LIN {X 0,Y 383.942,Z 862.362,A -85,B 0,C 180,E1 18991.194,E2 18991.194} C_VEL
LIN {X 0,Y 383.942,Z 862.362,A -85,B 0,C 180,E1 18988.806,E2 18988.806} C_VEL
LIN {X 0,Y 383.936,Z 861.248,A -85,B 0,C 180,E1 18986.267,E2 18986.267} C_VEL
LIN {X 0,Y 383.976,Z 858.254,A -85,B 0,C 180,E1 18983.121,E2 18983.121} C_VEL
LIN {X 0,Y 384.141,Z 854.129,A -85,B 0,C 180,E1 18980.411,E2 18980.411} C_VEL
LIN {X 0,Y 384.492,Z 848.967,A -85,B 0,C 180,E1 18977.841,E2 18977.841} C_VEL
LIN {X 0,Y 385.264,Z 841.518,A -85,B 0,C 180,E1 18974.901,E2 18974.901} C_VEL
LIN {X 0,Y 386.443,Z 832.341,A -85,B 0,C 180,E1 18972.068,E2 18972.068} C_VEL
LIN {X 0,Y 387.786,Z 823.59,A -85,B 0,C 180,E1 18969.788,E2 18969.788} C_VEL
LIN {X 0,Y 389.798,Z 811.997,A -85,B 0,C 180,E1 18967.213,E2 18967.213} C_VEL
LIN {X 0,Y 392.168,Z 798.843,A -85,B 0,C 180,E1 18964.801,E2 18964.801} C_VEL
LIN {X 0,Y 394.491,Z 786.516,A -85,B 0,C 180,E1 18962.857,E2 18962.857} C_VEL
LIN {X 0,Y 397.519,Z 770.561,A -85,B 0,C 180,E1 18960.712,E2 18960.712} C_VEL
LIN {X 0,Y 400.36,Z 754.684,A -85,B 0,C 180,E1 18958.943,E2 18958.943} C_VEL
LIN {X 0,Y 402.909,Z 739.928,A -85,B 0,C 180,E1 18957.543,E2 18957.543} C_VEL
LIN {X 0,Y 405.855,Z 721.57,A -85,B 0,C 180,E1 18956.083,E2 18956.083} C_VEL
LIN {X 0,Y 408.29,Z 703.761,A -85,B 0,C 180,E1 18954.953,E2 18954.953} C_VEL
LIN {X 0,Y 410.239,Z 687.519,A -85,B 0,C 180,E1 18954.116,E2 18954.116} C_VEL
LIN {X 0,Y 412.235,Z 667.836,A -85,B 0,C 180,E1 18953.326,E2 18953.326} C_VEL
LIN {X 0,Y 413.644,Z 647.128,A -85,B 0,C 180,E1 18952.766,E2 18952.766} C_VEL
LIN {X 0,Y 420.093,Z 444.232,A -85,B 0,C 180,E1 18949.037,E2 18949.037} C_VEL
LIN {X 0,Y 418.812,Z 440.206,A -85,B 0,C 180,E1 18948.796,E2 18948.796} C_VEL
LIN {X 0,Y 408.36,Z 420.188,A -85,B 0,C 180,E1 18947.041,E2 18947.041} C_VEL
LIN {X 0,Y 398.971,Z 403.892,A -85,B 0,C 180,E1 18945.381,E2 18945.381} C_VEL
LIN {X 0,Y 391.846,Z 392.481,A -85,B 0,C 180,E1 18944.058,E2 18944.058} C_VEL
LIN {X 0,Y 389.279,Z 388.042,A -85,B 0,C 180,E1 18943.505,E2 18943.505} C_VEL
LIN {X 0,Y 385.572,Z 377.041,A -85,B 0,C 180,E1 18940.395,E2 18940.395} C_VEL
LIN {X 0,Y 385.574,Z 376.942,A -85,B 0,C 180,E1 18936.619,E2 18936.619} C_VEL
LIN {X 0,Y 385.58,Z 376.931,A -85,B 0,C 180,E1 18932.646,E2 18932.646} C_VEL
LIN {X 0,Y 385.598,Z 376.915,A -85,B 0,C 180,E1 18928.788,E2 18928.788} C_VEL
LIN {X 0,Y 385.593,Z 376.956,A -85,B 0,C 180,E1 18924.681,E2 18924.681} C_VEL
LIN {X 0,Y 385.592,Z 376.909,A -85,B 0,C 180,E1 18920.655,E2 18920.655} C_VEL
LIN {X 0,Y 385.593,Z 376.941,A -85,B 0,C 180,E1 18916.578,E2 18916.578} C_VEL
LIN {X 0,Y 385.593,Z 376.919,A -85,B 0,C 180,E1 18912.586,E2 18912.586} C_VEL
LIN {X 0,Y 385.597,Z 376.93,A -85,B 0,C 180,E1 18908.505,E2 18908.505} C_VEL
LIN {X 0,Y 385.591,Z 376.927,A -85,B 0,C 180,E1 18904.468,E2 18904.468} C_VEL
LIN {X 0,Y 385.605,Z 376.925,A -85,B 0,C 180,E1 18900.452,E2 18900.452} C_VEL
LIN {X 0,Y 385.591,Z 376.927,A -85,B 0,C 180,E1 18896.439,E2 18896.439} C_VEL
LIN {X 0,Y 385.601,Z 376.923,A -85,B 0,C 180,E1 18892.408,E2 18892.408} C_VEL
LIN {X 0,Y 385.592,Z 376.934,A -85,B 0,C 180,E1 18888.338,E2 18888.338} C_VEL
LIN {X 0,Y 385.589,Z 376.916,A -85,B 0,C 180,E1 18884.363,E2 18884.363} C_VEL
LIN {X 0,Y 385.595,Z 376.946,A -85,B 0,C 180,E1 18880.261,E2 18880.261} C_VEL
LIN {X 0,Y 385.581,Z 376.911,A -85,B 0,C 180,E1 18876.31,E2 18876.31} C_VEL
LIN {X 0,Y 385.578,Z 376.958,A -85,B 0,C 180,E1 18872.353,E2 18872.353} C_VEL
LIN {X 0,Y 385.562,Z 376.958,A -85,B 0,C 180,E1 18868.556,E2 18868.556} C_VEL
LIN {X 0,Y 385.554,Z 376.96,A -85,B 0,C 180,E1 18864.679,E2 18864.679} C_VEL
LIN {X 0,Y 385.55,Z 376.957,A -85,B 0,C 180,E1 18860.757,E2 18860.757} C_VEL
LIN {X 0,Y 385.553,Z 376.96,A -85,B 0,C 180,E1 18856.777,E2 18856.777} C_VEL
LIN {X 0,Y 385.553,Z 376.96,A -85,B 0,C 180,E1 18852.799,E2 18852.799} C_VEL
LIN {X 0,Y 385.554,Z 376.956,A -85,B 0,C 180,E1 18848.87,E2 18848.87} C_VEL
LIN {X 0,Y 385.56,Z 376.957,A -85,B 0,C 180,E1 18844.966,E2 18844.966} C_VEL
LIN {X 0,Y 385.568,Z 376.959,A -85,B 0,C 180,E1 18841.067,E2 18841.067} C_VEL
LIN {X 0,Y 385.579,Z 376.954,A -85,B 0,C 180,E1 18837.154,E2 18837.154} C_VEL
LIN {X 0,Y 385.628,Z 377.162,A -85,B 0,C 180,E1 18833.371,E2 18833.371} C_VEL
LIN {X 0,Y 386.073,Z 378.926,A -85,B 0,C 180,E1 18831.816,E2 18831.816} C_VEL
LIN {X 0,Y 387.404,Z 381.16,A -85,B 0,C 180,E1 18830.07,E2 18830.07} C_VEL
LIN {X 0,Y 389.591,Z 382.927,A -85,B 0,C 180,E1 18827.165,E2 18827.165} C_VEL
LIN {X 0,Y 391.833,Z 384.088,A -85,B 0,C 180,E1 18823.728,E2 18823.728} C_VEL
LIN {X 0,Y 393.13,Z 386.138,A -85,B 0,C 180,E1 18820.996,E2 18820.996} C_VEL
LIN {X 0,Y 394.172,Z 387.9,A -85,B 0,C 180,E1 18818.166,E2 18818.166} C_VEL
LIN {X 0,Y 395.064,Z 388.811,A -85,B 0,C 180,E1 18814.791,E2 18814.791} C_VEL
LIN {X 0,Y 395.484,Z 389.178,A -85,B 0,C 180,E1 18811.449,E2 18811.449} C_VEL
LIN {X 0,Y 395.444,Z 389.163,A -85,B 0,C 180,E1 18808.116,E2 18808.116} C_VEL
LIN {X 0,Y 394.988,Z 388.728,A -85,B 0,C 180,E1 18804.917,E2 18804.917} C_VEL
LIN {X 0,Y 394.109,Z 387.826,A -85,B 0,C 180,E1 18801.686,E2 18801.686} C_VEL
LIN {X 0,Y 393.123,Z 386.118,A -85,B 0,C 180,E1 18798.98,E2 18798.98} C_VEL
LIN {X 0,Y 391.832,Z 384.088,A -85,B 0,C 180,E1 18796.272,E2 18796.272} C_VEL
LIN {X 0,Y 389.591,Z 382.928,A -85,B 0,C 180,E1 18792.835,E2 18792.835} C_VEL
LIN {X 0,Y 387.4,Z 381.156,A -85,B 0,C 180,E1 18789.925,E2 18789.925} C_VEL
LIN {X 0,Y 386.016,Z 378.794,A -85,B 0,C 180,E1 18788.101,E2 18788.101} C_VEL
LIN {X 0,Y 385.613,Z 377.094,A -85,B 0,C 180,E1 18786.51,E2 18786.51} C_VEL
LIN {X 0,Y 385.593,Z 376.953,A -85,B 0,C 180,E1 18782.651,E2 18782.651} C_VEL
LIN {X 0,Y 384.623,Z 377.077,A -85,B 0,C 180,E1 18781.507,E2 18781.507} C_VEL
LIN {X 0,Y 379.656,Z 377.695,A -85,B 0,C 180,E1 18779.185,E2 18779.185} C_VEL
LIN {X 0,Y 377.705,Z 377.936,A -85,B 0,C 180,E1 18777.774,E2 18777.774} C_VEL
LIN {X 0,Y 377.612,Z 377.948,A -85,B 0,C 180,E1 18777.434,E2 18777.434} C_VEL
LIN {X 0,Y 377.613,Z 377.947,A -85,B 0,C 180,E1 18773.333,E2 18773.333} C_VEL
LIN {X 0,Y 377.611,Z 377.946,A -85,B 0,C 180,E1 18769.356,E2 18769.356} C_VEL
LIN {X 0,Y 377.613,Z 377.95,A -85,B 0,C 180,E1 18765.227,E2 18765.227} C_VEL
LIN {X 0,Y 377.612,Z 377.947,A -85,B 0,C 180,E1 18761.235,E2 18761.235} C_VEL
LIN {X 0,Y 377.615,Z 377.945,A -85,B 0,C 180,E1 18757.124,E2 18757.124} C_VEL
LIN {X 0,Y 377.614,Z 377.949,A -85,B 0,C 180,E1 18753.045,E2 18753.045} C_VEL
LIN {X 0,Y 377.616,Z 377.947,A -85,B 0,C 180,E1 18748.973,E2 18748.973} C_VEL
LIN {X 0,Y 377.61,Z 377.907,A -85,B 0,C 180,E1 18744.889,E2 18744.889} C_VEL
LIN {X 0,Y 377.615,Z 377.947,A -85,B 0,C 180,E1 18740.773,E2 18740.773} C_VEL
LIN {X 0,Y 377.608,Z 377.895,A -85,B 0,C 180,E1 18736.767,E2 18736.767} C_VEL
LIN {X 0,Y 377.613,Z 377.947,A -85,B 0,C 180,E1 18732.688,E2 18732.688} C_VEL
LIN {X 0,Y 377.609,Z 377.896,A -85,B 0,C 180,E1 18728.673,E2 18728.673} C_VEL
LIN {X 0,Y 377.615,Z 377.94,A -85,B 0,C 180,E1 18724.549,E2 18724.549} C_VEL
LIN {X 0,Y 377.609,Z 377.899,A -85,B 0,C 180,E1 18720.449,E2 18720.449} C_VEL
LIN {X 0,Y 377.614,Z 377.941,A -85,B 0,C 180,E1 18716.502,E2 18716.502} C_VEL
LIN {X 0,Y 377.609,Z 377.901,A -85,B 0,C 180,E1 18712.386,E2 18712.386} C_VEL
LIN {X 0,Y 377.616,Z 377.933,A -85,B 0,C 180,E1 18708.385,E2 18708.385} C_VEL
LIN {X 0,Y 377.614,Z 377.91,A -85,B 0,C 180,E1 18704.325,E2 18704.325} C_VEL
LIN {X 0,Y 377.615,Z 377.918,A -85,B 0,C 180,E1 18700.344,E2 18700.344} C_VEL
LIN {X 0,Y 377.617,Z 377.936,A -85,B 0,C 180,E1 18696.262,E2 18696.262} C_VEL
LIN {X 0,Y 377.613,Z 377.902,A -85,B 0,C 180,E1 18692.172,E2 18692.172} C_VEL
LIN {X 0,Y 377.621,Z 377.935,A -85,B 0,C 180,E1 18688.198,E2 18688.198} C_VEL
LIN {X 0,Y 377.62,Z 377.947,A -85,B 0,C 180,E1 18684.115,E2 18684.115} C_VEL
LIN {X 0,Y 377.681,Z 378.167,A -85,B 0,C 180,E1 18680.625,E2 18680.625} C_VEL
LIN {X 0,Y 381.123,Z 388.069,A -85,B 0,C 180,E1 18677.756,E2 18677.756} C_VEL
LIN {X 0,Y 390.405,Z 402.884,A -85,B 0,C 180,E1 18675.89,E2 18675.89} C_VEL
LIN {X 0,Y 399.613,Z 418.325,A -85,B 0,C 180,E1 18674.175,E2 18674.175} C_VEL
LIN {X 0,Y 409.795,Z 437.296,A -85,B 0,C 180,E1 18672.376,E2 18672.376} C_VEL
LIN {X 0,Y 414.001,Z 446.197,A -85,B 0,C 180,E1 18671.649,E2 18671.649} C_VEL
LIN {X 0,Y 407.264,Z 647.302,A -85,B 0,C 180,E1 18667.908,E2 18667.908} C_VEL
LIN {X 0,Y 405.749,Z 668.252,A -85,B 0,C 180,E1 18667.327,E2 18667.327} C_VEL
LIN {X 0,Y 403.735,Z 687.281,A -85,B 0,C 180,E1 18666.554,E2 18666.554} C_VEL
LIN {X 0,Y 401.698,Z 703.522,A -85,B 0,C 180,E1 18665.709,E2 18665.709} C_VEL
LIN {X 0,Y 399,Z 722.359,A -85,B 0,C 180,E1 18664.494,E2 18664.494} C_VEL
LIN {X 0,Y 395.936,Z 740.419,A -85,B 0,C 180,E1 18663.023,E2 18663.023} C_VEL
LIN {X 0,Y 393.241,Z 755.268,A -85,B 0,C 180,E1 18661.585,E2 18661.585} C_VEL
LIN {X 0,Y 390.053,Z 772.125,A -85,B 0,C 180,E1 18659.651,E2 18659.651} C_VEL
LIN {X 0,Y 387.116,Z 786.716,A -85,B 0,C 180,E1 18657.63,E2 18657.63} C_VEL
LIN {X 0,Y 384.752,Z 798.6,A -85,B 0,C 180,E1 18655.72,E2 18655.72} C_VEL
LIN {X 0,Y 382.233,Z 811.754,A -85,B 0,C 180,E1 18653.265,E2 18653.265} C_VEL
LIN {X 0,Y 380.084,Z 823.347,A -85,B 0,C 180,E1 18650.64,E2 18650.64} C_VEL
LIN {X 0,Y 378.649,Z 832.099,A -85,B 0,C 180,E1 18648.314,E2 18648.314} C_VEL
LIN {X 0,Y 377.41,Z 840.984,A -85,B 0,C 180,E1 18645.52,E2 18645.52} C_VEL
LIN {X 0,Y 376.575,Z 848.391,A -85,B 0,C 180,E1 18642.575,E2 18642.575} C_VEL
LIN {X 0,Y 376.174,Z 853.618,A -85,B 0,C 180,E1 18639.948,E2 18639.948} C_VEL
LIN {X 0,Y 375.996,Z 857.669,A -85,B 0,C 180,E1 18637.281,E2 18637.281} C_VEL
LIN {X 0,Y 375.934,Z 860.833,A -85,B 0,C 180,E1 18634.118,E2 18634.118} C_VEL
LIN {X 0,Y 375.941,Z 862.096,A -85,B 0,C 180,E1 18631.372,E2 18631.372} C_VEL
LIN {X 0,Y 375.946,Z 862.156,A -85,B 0,C 180,E1 18628.933,E2 18628.933} C_VEL
LIN {X 0,Y 375.939,Z 861.189,A -85,B 0,C 180,E1 18626.493,E2 18626.493} C_VEL
LIN {X 0,Y 375.956,Z 858.89,A -85,B 0,C 180,E1 18623.74,E2 18623.74} C_VEL
LIN {X 0,Y 376.132,Z 854.392,A -85,B 0,C 180,E1 18620.491,E2 18620.491} C_VEL
LIN {X 0,Y 376.484,Z 849.397,A -85,B 0,C 180,E1 18617.889,E2 18617.889} C_VEL
LIN {X 0,Y 377.146,Z 843.059,A -85,B 0,C 180,E1 18615.256,E2 18615.256} C_VEL
LIN {X 0,Y 378.408,Z 833.73,A -85,B 0,C 180,E1 18612.152,E2 18612.152} C_VEL
LIN {X 0,Y 379.871,Z 824.59,A -85,B 0,C 180,E1 18609.67,E2 18609.67} C_VEL
LIN {X 0,Y 381.668,Z 814.59,A -85,B 0,C 180,E1 18607.351,E2 18607.351} C_VEL
LIN {X 0,Y 384.239,Z 801.279,A -85,B 0,C 180,E1 18604.739,E2 18604.739} C_VEL
LIN {X 0,Y 386.807,Z 788.278,A -85,B 0,C 180,E1 18602.607,E2 18602.607} C_VEL
LIN {X 0,Y 389.346,Z 775.499,A -85,B 0,C 180,E1 18600.796,E2 18600.796} C_VEL
LIN {X 0,Y 392.617,Z 758.832,A -85,B 0,C 180,E1 18598.787,E2 18598.787} C_VEL
LIN {X 0,Y 395.564,Z 742.542,A -85,B 0,C 180,E1 18597.168,E2 18597.168} C_VEL
LIN {X 0,Y 398.2,Z 726.983,A -85,B 0,C 180,E1 18595.863,E2 18595.863} C_VEL
LIN {X 0,Y 401.068,Z 708.502,A -85,B 0,C 180,E1 18594.578,E2 18594.578} C_VEL
LIN {X 0,Y 403.508,Z 689.272,A -85,B 0,C 180,E1 18593.54,E2 18593.54} C_VEL
LIN {X 0,Y 405.339,Z 672.186,A -85,B 0,C 180,E1 18592.819,E2 18592.819} C_VEL
LIN {X 0,Y 407.074,Z 651.206,A -85,B 0,C 180,E1 18592.177,E2 18592.177} C_VEL
LIN {X 0,Y 408.543,Z 611.703,A -85,B 0,C 180,E1 18591.406,E2 18591.406} C_VEL
LIN {X 0,Y 413.876,Z 445.539,A -85,B 0,C 180,E1 18588.321,E2 18588.321} C_VEL
LIN {X 0,Y 403.611,Z 425.576,A -85,B 0,C 180,E1 18586.544,E2 18586.544} C_VEL
LIN {X 0,Y 394.17,Z 409.047,A -85,B 0,C 180,E1 18584.823,E2 18584.823} C_VEL
LIN {X 0,Y 387.437,Z 398.145,A -85,B 0,C 180,E1 18583.534,E2 18583.534} C_VEL
LIN {X 0,Y 380.95,Z 387.635,A -85,B 0,C 180,E1 18582.169,E2 18582.169} C_VEL
LIN {X 0,Y 377.669,Z 378.032,A -85,B 0,C 180,E1 18579.288,E2 18579.288} C_VEL
LIN {X 0,Y 377.652,Z 377.94,A -85,B 0,C 180,E1 18575.257,E2 18575.257} C_VEL
LIN {X 0,Y 377.651,Z 377.942,A -85,B 0,C 180,E1 18571.225,E2 18571.225} C_VEL
LIN {X 0,Y 377.646,Z 377.902,A -85,B 0,C 180,E1 18567.181,E2 18567.181} C_VEL
LIN {X 0,Y 377.636,Z 377.921,A -85,B 0,C 180,E1 18563.24,E2 18563.24} C_VEL
LIN {X 0,Y 377.628,Z 377.925,A -85,B 0,C 180,E1 18559.333,E2 18559.333} C_VEL
LIN {X 0,Y 377.619,Z 377.903,A -85,B 0,C 180,E1 18555.36,E2 18555.36} C_VEL
LIN {X 0,Y 377.618,Z 377.938,A -85,B 0,C 180,E1 18551.46,E2 18551.46} C_VEL
LIN {X 0,Y 377.61,Z 377.899,A -85,B 0,C 180,E1 18547.461,E2 18547.461} C_VEL
LIN {X 0,Y 377.614,Z 377.942,A -85,B 0,C 180,E1 18543.437,E2 18543.437} C_VEL
LIN {X 0,Y 377.609,Z 377.897,A -85,B 0,C 180,E1 18539.4,E2 18539.4} C_VEL
LIN {X 0,Y 377.616,Z 377.943,A -85,B 0,C 180,E1 18535.299,E2 18535.299} C_VEL
LIN {X 0,Y 377.609,Z 377.896,A -85,B 0,C 180,E1 18531.327,E2 18531.327} C_VEL
LIN {X 0,Y 377.613,Z 377.947,A -85,B 0,C 180,E1 18527.312,E2 18527.312} C_VEL
LIN {X 0,Y 377.608,Z 377.895,A -85,B 0,C 180,E1 18523.233,E2 18523.233} C_VEL
LIN {X 0,Y 377.614,Z 377.947,A -85,B 0,C 180,E1 18519.173,E2 18519.173} C_VEL
LIN {X 0,Y 377.61,Z 377.907,A -85,B 0,C 180,E1 18515.111,E2 18515.111} C_VEL
LIN {X 0,Y 377.616,Z 377.947,A -85,B 0,C 180,E1 18511.027,E2 18511.027} C_VEL
LIN {X 0,Y 377.614,Z 377.949,A -85,B 0,C 180,E1 18506.955,E2 18506.955} C_VEL
LIN {X 0,Y 377.616,Z 377.945,A -85,B 0,C 180,E1 18502.842,E2 18502.842} C_VEL
LIN {X 0,Y 377.612,Z 377.947,A -85,B 0,C 180,E1 18498.761,E2 18498.761} C_VEL
LIN {X 0,Y 377.613,Z 377.95,A -85,B 0,C 180,E1 18494.773,E2 18494.773} C_VEL
LIN {X 0,Y 377.611,Z 377.946,A -85,B 0,C 180,E1 18490.644,E2 18490.644} C_VEL
LIN {X 0,Y 377.612,Z 377.947,A -85,B 0,C 180,E1 18486.566,E2 18486.566} C_VEL
LIN {X 0,Y 377.613,Z 377.948,A -85,B 0,C 180,E1 18482.513,E2 18482.513} C_VEL
LIN {X 0,Y 377.672,Z 378.275,A -85,B 0,C 180,E1 18480.023,E2 18480.023} C_VEL
LIN {X 0,Y 378.13,Z 379.915,A -85,B 0,C 180,E1 18478.939,E2 18478.939} C_VEL
LIN {X 0,Y 379.727,Z 382.394,A -85,B 0,C 180,E1 18477.352,E2 18477.352} C_VEL
LIN {X 0,Y 382.065,Z 384.142,A -85,B 0,C 180,E1 18475.084,E2 18475.084} C_VEL
LIN {X 0,Y 384.206,Z 385.45,A -85,B 0,C 180,E1 18472.917,E2 18472.917} C_VEL
LIN {X 0,Y 386.14,Z 388.832,A -85,B 0,C 180,E1 18470.419,E2 18470.419} C_VEL
LIN {X 0,Y 388.364,Z 390.735,A -85,B 0,C 180,E1 18467.53,E2 18467.53} C_VEL
LIN {X 0,Y 390.583,Z 391.827,A -85,B 0,C 180,E1 18464.226,E2 18464.226} C_VEL
LIN {X 0,Y 391.743,Z 393.325,A -85,B 0,C 180,E1 18461.931,E2 18461.931} C_VEL
LIN {X 0,Y 392.813,Z 395.259,A -85,B 0,C 180,E1 18459.227,E2 18459.227} C_VEL
LIN {X 0,Y 393.737,Z 396.441,A -85,B 0,C 180,E1 18456.269,E2 18456.269} C_VEL
LIN {X 0,Y 394.362,Z 396.976,A -85,B 0,C 180,E1 18453.052,E2 18453.052} C_VEL
LIN {X 0,Y 394.538,Z 397.156,A -85,B 0,C 180,E1 18449.71,E2 18449.71} C_VEL
LIN {X 0,Y 394.293,Z 396.941,A -85,B 0,C 180,E1 18446.511,E2 18446.511} C_VEL
LIN {X 0,Y 393.6,Z 396.299,A -85,B 0,C 180,E1 18443.252,E2 18443.252} C_VEL
LIN {X 0,Y 392.612,Z 395.021,A -85,B 0,C 180,E1 18440.176,E2 18440.176} C_VEL
LIN {X 0,Y 391.176,Z 392.348,A -85,B 0,C 180,E1 18436.822,E2 18436.822} C_VEL
LIN {X 0,Y 389.393,Z 391.283,A -85,B 0,C 180,E1 18433.9,E2 18433.9} C_VEL
LIN {X 0,Y 387.152,Z 389.847,A -85,B 0,C 180,E1 18430.854,E2 18430.854} C_VEL
LIN {X 0,Y 385.342,Z 387.618,A -85,B 0,C 180,E1 18428.54,E2 18428.54} C_VEL
LIN {X 0,Y 383.815,Z 385.017,A -85,B 0,C 180,E1 18426.674,E2 18426.674} C_VEL
LIN {X 0,Y 380.576,Z 383.223,A -85,B 0,C 180,E1 18423.473,E2 18423.473} C_VEL
LIN {X 0,Y 378.591,Z 380.901,A -85,B 0,C 180,E1 18421.555,E2 18421.555} C_VEL
LIN {X 0,Y 377.728,Z 378.489,A -85,B 0,C 180,E1 18420.233,E2 18420.233} C_VEL
LIN {X 0,Y 377.657,Z 377.942,A -85,B 0,C 180,E1 18418.564,E2 18418.564} C_VEL
LIN {X 0,Y 377.612,Z 377.948,A -85,B 0,C 180,E1 18417.434,E2 18417.434} C_VEL
LIN {X 0,Y 376.644,Z 378.078,A -85,B 0,C 180,E1 18416.266,E2 18416.266} C_VEL
LIN {X 0,Y 371.769,Z 378.689,A -85,B 0,C 180,E1 18413.892,E2 18413.892} C_VEL
LIN {X 0,Y 369.813,Z 378.925,A -85,B 0,C 180,E1 18412.45,E2 18412.45} C_VEL
LIN {X 0,Y 369.702,Z 378.936,A -85,B 0,C 180,E1 18412.104,E2 18412.104} C_VEL
LIN {X 0,Y 369.706,Z 378.931,A -85,B 0,C 180,E1 18408.035,E2 18408.035} C_VEL
LIN {X 0,Y 369.704,Z 378.932,A -85,B 0,C 180,E1 18403.997,E2 18403.997} C_VEL
LIN {X 0,Y 369.717,Z 378.933,A -85,B 0,C 180,E1 18400.052,E2 18400.052} C_VEL
LIN {X 0,Y 369.708,Z 378.934,A -85,B 0,C 180,E1 18395.924,E2 18395.924} C_VEL
LIN {X 0,Y 369.708,Z 378.935,A -85,B 0,C 180,E1 18391.817,E2 18391.817} C_VEL
LIN {X 0,Y 369.716,Z 378.933,A -85,B 0,C 180,E1 18387.833,E2 18387.833} C_VEL
LIN {X 0,Y 369.707,Z 378.884,A -85,B 0,C 180,E1 18383.754,E2 18383.754} C_VEL
LIN {X 0,Y 369.715,Z 378.923,A -85,B 0,C 180,E1 18379.749,E2 18379.749} C_VEL
LIN {X 0,Y 369.713,Z 378.889,A -85,B 0,C 180,E1 18375.682,E2 18375.682} C_VEL
LIN {X 0,Y 369.713,Z 378.909,A -85,B 0,C 180,E1 18371.695,E2 18371.695} C_VEL
LIN {X 0,Y 369.723,Z 378.896,A -85,B 0,C 180,E1 18367.607,E2 18367.607} C_VEL
LIN {X 0,Y 369.711,Z 378.9,A -85,B 0,C 180,E1 18363.559,E2 18363.559} C_VEL
LIN {X 0,Y 369.715,Z 378.905,A -85,B 0,C 180,E1 18359.373,E2 18359.373} C_VEL
LIN {X 0,Y 369.71,Z 378.895,A -85,B 0,C 180,E1 18355.34,E2 18355.34} C_VEL
LIN {X 0,Y 369.716,Z 378.909,A -85,B 0,C 180,E1 18351.283,E2 18351.283} C_VEL
LIN {X 0,Y 369.71,Z 378.888,A -85,B 0,C 180,E1 18347.181,E2 18347.181} C_VEL
LIN {X 0,Y 369.716,Z 378.921,A -85,B 0,C 180,E1 18343.174,E2 18343.174} C_VEL
LIN {X 0,Y 369.715,Z 378.881,A -85,B 0,C 180,E1 18339.079,E2 18339.079} C_VEL
LIN {X 0,Y 369.716,Z 378.931,A -85,B 0,C 180,E1 18334.951,E2 18334.951} C_VEL
LIN {X 0,Y 369.713,Z 378.896,A -85,B 0,C 180,E1 18330.864,E2 18330.864} C_VEL
LIN {X 0,Y 369.716,Z 378.902,A -85,B 0,C 180,E1 18326.882,E2 18326.882} C_VEL
LIN {X 0,Y 369.717,Z 378.909,A -85,B 0,C 180,E1 18322.904,E2 18322.904} C_VEL
LIN {X 0,Y 369.726,Z 379.233,A -85,B 0,C 180,E1 18321.763,E2 18321.763} C_VEL
LIN {X 0,Y 372.748,Z 387.649,A -85,B 0,C 180,E1 18319.195,E2 18319.195} C_VEL
LIN {X 0,Y 376.572,Z 393.398,A -85,B 0,C 180,E1 18318.354,E2 18318.354} C_VEL
LIN {X 0,Y 386.522,Z 409.416,A -85,B 0,C 180,E1 18316.311,E2 18316.311} C_VEL
LIN {X 0,Y 395.558,Z 424.826,A -85,B 0,C 180,E1 18314.582,E2 18314.582} C_VEL
LIN {X 0,Y 406.274,Z 445.199,A -85,B 0,C 180,E1 18312.642,E2 18312.642} C_VEL
LIN {X 0,Y 407.925,Z 449.067,A -85,B 0,C 180,E1 18312.34,E2 18312.34} C_VEL
LIN {X 0,Y 400.962,Z 647.065,A -85,B 0,C 180,E1 18308.613,E2 18308.613} C_VEL
LIN {X 0,Y 399.38,Z 668.11,A -85,B 0,C 180,E1 18308.022,E2 18308.022} C_VEL
LIN {X 0,Y 397.291,Z 687.043,A -85,B 0,C 180,E1 18307.247,E2 18307.247} C_VEL
LIN {X 0,Y 395.088,Z 703.844,A -85,B 0,C 180,E1 18306.361,E2 18306.361} C_VEL
LIN {X 0,Y 392.085,Z 723.574,A -85,B 0,C 180,E1 18305.052,E2 18305.052} C_VEL
LIN {X 0,Y 389.199,Z 739.878,A -85,B 0,C 180,E1 18303.703,E2 18303.703} C_VEL
LIN {X 0,Y 386.313,Z 755.027,A -85,B 0,C 180,E1 18302.219,E2 18302.219} C_VEL
LIN {X 0,Y 382.965,Z 771.884,A -85,B 0,C 180,E1 18300.257,E2 18300.257} C_VEL
LIN {X 0,Y 379.851,Z 786.532,A -85,B 0,C 180,E1 18298.195,E2 18298.195} C_VEL
LIN {X 0,Y 377.367,Z 798.358,A -85,B 0,C 180,E1 18296.261,E2 18296.261} C_VEL
LIN {X 0,Y 374.669,Z 811.622,A -85,B 0,C 180,E1 18293.738,E2 18293.738} C_VEL
LIN {X 0,Y 372.407,Z 823.104,A -85,B 0,C 180,E1 18291.085,E2 18291.085} C_VEL
LIN {X 0,Y 370.87,Z 831.857,A -85,B 0,C 180,E1 18288.712,E2 18288.712} C_VEL
LIN {X 0,Y 369.536,Z 840.743,A -85,B 0,C 180,E1 18285.859,E2 18285.859} C_VEL
LIN {X 0,Y 368.635,Z 848.151,A -85,B 0,C 180,E1 18282.85,E2 18282.85} C_VEL
LIN {X 0,Y 368.194,Z 853.378,A -85,B 0,C 180,E1 18280.166,E2 18280.166} C_VEL
LIN {X 0,Y 368.005,Z 857.359,A -85,B 0,C 180,E1 18277.493,E2 18277.493} C_VEL
LIN {X 0,Y 367.934,Z 860.623,A -85,B 0,C 180,E1 18274.161,E2 18274.161} C_VEL
LIN {X 0,Y 367.944,Z 861.86,A -85,B 0,C 180,E1 18271.401,E2 18271.401} C_VEL
LIN {X 0,Y 367.949,Z 861.919,A -85,B 0,C 180,E1 18268.91,E2 18268.91} C_VEL
LIN {X 0,Y 367.941,Z 860.952,A -85,B 0,C 180,E1 18266.417,E2 18266.417} C_VEL
LIN {X 0,Y 367.958,Z 858.652,A -85,B 0,C 180,E1 18263.604,E2 18263.604} C_VEL
LIN {X 0,Y 368.15,Z 854.193,A -85,B 0,C 180,E1 18260.306,E2 18260.306} C_VEL
LIN {X 0,Y 368.536,Z 849.149,A -85,B 0,C 180,E1 18257.62,E2 18257.62} C_VEL
LIN {X 0,Y 369.253,Z 842.818,A -85,B 0,C 180,E1 18254.934,E2 18254.934} C_VEL
LIN {X 0,Y 370.622,Z 833.424,A -85,B 0,C 180,E1 18251.745,E2 18251.745} C_VEL
LIN {X 0,Y 372.186,Z 824.295,A -85,B 0,C 180,E1 18249.217,E2 18249.217} C_VEL
LIN {X 0,Y 374.119,Z 814.233,A -85,B 0,C 180,E1 18246.841,E2 18246.841} C_VEL
LIN {X 0,Y 377.018,Z 800.074,A -85,B 0,C 180,E1 18244.038,E2 18244.038} C_VEL
LIN {X 0,Y 379.713,Z 787.184,A -85,B 0,C 180,E1 18241.905,E2 18241.905} C_VEL
LIN {X 0,Y 382.713,Z 773.008,A -85,B 0,C 180,E1 18239.894,E2 18239.894} C_VEL
LIN {X 0,Y 386.187,Z 755.695,A -85,B 0,C 180,E1 18237.851,E2 18237.851} C_VEL
LIN {X 0,Y 389.011,Z 740.888,A -85,B 0,C 180,E1 18236.389,E2 18236.389} C_VEL
LIN {X 0,Y 391.845,Z 724.899,A -85,B 0,C 180,E1 18235.052,E2 18235.052} C_VEL
LIN {X 0,Y 394.996,Z 704.529,A -85,B 0,C 180,E1 18233.679,E2 18233.679} C_VEL
LIN {X 0,Y 397.2,Z 687.787,A -85,B 0,C 180,E1 18232.789,E2 18232.789} C_VEL
LIN {X 0,Y 399.207,Z 669.659,A -85,B 0,C 180,E1 18232.035,E2 18232.035} C_VEL
LIN {X 0,Y 400.925,Z 647.784,A -85,B 0,C 180,E1 18231.403,E2 18231.403} C_VEL
LIN {X 0,Y 404.208,Z 555.001,A -85,B 0,C 180,E1 18229.639,E2 18229.639} C_VEL
LIN {X 0,Y 407.785,Z 448.372,A -85,B 0,C 180,E1 18227.626,E2 18227.626} C_VEL
LIN {X 0,Y 398.188,Z 429.718,A -85,B 0,C 180,E1 18225.907,E2 18225.907} C_VEL
LIN {X 0,Y 389.274,Z 413.969,A -85,B 0,C 180,E1 18224.226,E2 18224.226} C_VEL
LIN {X 0,Y 382.536,Z 402.995,A -85,B 0,C 180,E1 18222.892,E2 18222.892} C_VEL
LIN {X 0,Y 375.82,Z 392.518,A -85,B 0,C 180,E1 18221.493,E2 18221.493} C_VEL
LIN {X 0,Y 372.52,Z 387.202,A -85,B 0,C 180,E1 18220.715,E2 18220.715} C_VEL
LIN {X 0,Y 369.69,Z 379.011,A -85,B 0,C 180,E1 18218.121,E2 18218.121} C_VEL
LIN {X 0,Y 369.677,Z 378.91,A -85,B 0,C 180,E1 18214.052,E2 18214.052} C_VEL
LIN {X 0,Y 369.68,Z 378.922,A -85,B 0,C 180,E1 18210.029,E2 18210.029} C_VEL
LIN {X 0,Y 369.68,Z 378.919,A -85,B 0,C 180,E1 18205.819,E2 18205.819} C_VEL
LIN {X 0,Y 369.676,Z 378.886,A -85,B 0,C 180,E1 18201.755,E2 18201.755} C_VEL
LIN {X 0,Y 369.678,Z 378.936,A -85,B 0,C 180,E1 18197.639,E2 18197.639} C_VEL
LIN {X 0,Y 369.672,Z 378.882,A -85,B 0,C 180,E1 18193.616,E2 18193.616} C_VEL
LIN {X 0,Y 369.678,Z 378.931,A -85,B 0,C 180,E1 18189.503,E2 18189.503} C_VEL
LIN {X 0,Y 369.672,Z 378.885,A -85,B 0,C 180,E1 18185.438,E2 18185.438} C_VEL
LIN {X 0,Y 369.677,Z 378.927,A -85,B 0,C 180,E1 18181.401,E2 18181.401} C_VEL
LIN {X 0,Y 369.67,Z 378.885,A -85,B 0,C 180,E1 18177.372,E2 18177.372} C_VEL
LIN {X 0,Y 369.673,Z 378.925,A -85,B 0,C 180,E1 18173.329,E2 18173.329} C_VEL
LIN {X 0,Y 369.671,Z 378.891,A -85,B 0,C 180,E1 18169.252,E2 18169.252} C_VEL
LIN {X 0,Y 369.672,Z 378.918,A -85,B 0,C 180,E1 18165.279,E2 18165.279} C_VEL
LIN {X 0,Y 369.672,Z 378.903,A -85,B 0,C 180,E1 18161.195,E2 18161.195} C_VEL
LIN {X 0,Y 369.67,Z 378.897,A -85,B 0,C 180,E1 18157.087,E2 18157.087} C_VEL
LIN {X 0,Y 369.677,Z 378.937,A -85,B 0,C 180,E1 18152.984,E2 18152.984} C_VEL
LIN {X 0,Y 369.676,Z 378.937,A -85,B 0,C 180,E1 18148.906,E2 18148.906} C_VEL
LIN {X 0,Y 369.677,Z 378.938,A -85,B 0,C 180,E1 18144.765,E2 18144.765} C_VEL
LIN {X 0,Y 369.674,Z 378.935,A -85,B 0,C 180,E1 18140.671,E2 18140.671} C_VEL
LIN {X 0,Y 369.676,Z 378.938,A -85,B 0,C 180,E1 18136.621,E2 18136.621} C_VEL
LIN {X 0,Y 369.675,Z 378.935,A -85,B 0,C 180,E1 18132.544,E2 18132.544} C_VEL
LIN {X 0,Y 369.673,Z 378.935,A -85,B 0,C 180,E1 18128.467,E2 18128.467} C_VEL
LIN {X 0,Y 369.754,Z 379.246,A -85,B 0,C 180,E1 18125.737,E2 18125.737} C_VEL
LIN {X 0,Y 370.079,Z 380.623,A -85,B 0,C 180,E1 18124.9,E2 18124.9} C_VEL
LIN {X 0,Y 371.296,Z 382.818,A -85,B 0,C 180,E1 18123.826,E2 18123.826} C_VEL
LIN {X 0,Y 373.577,Z 384.842,A -85,B 0,C 180,E1 18121.978,E2 18121.978} C_VEL
LIN {X 0,Y 376.235,Z 386.428,A -85,B 0,C 180,E1 18119.798,E2 18119.798} C_VEL
LIN {X 0,Y 378.164,Z 389.818,A -85,B 0,C 180,E1 18117.903,E2 18117.903} C_VEL
LIN {X 0,Y 380.734,Z 391.911,A -85,B 0,C 180,E1 18115.417,E2 18115.417} C_VEL
LIN {X 0,Y 382.92,Z 393.129,A -85,B 0,C 180,E1 18113.22,E2 18113.22} C_VEL
LIN {X 0,Y 384.953,Z 396.576,A -85,B 0,C 180,E1 18110.685,E2 18110.685} C_VEL
LIN {X 0,Y 387.258,Z 398.614,A -85,B 0,C 180,E1 18107.723,E2 18107.723} C_VEL
LIN {X 0,Y 389.508,Z 399.699,A -85,B 0,C 180,E1 18104.418,E2 18104.418} C_VEL
LIN {X 0,Y 390.677,Z 401.156,A -85,B 0,C 180,E1 18102.114,E2 18102.114} C_VEL
LIN {X 0,Y 391.784,Z 403.135,A -85,B 0,C 180,E1 18099.4,E2 18099.4} C_VEL
LIN {X 0,Y 392.734,Z 404.354,A -85,B 0,C 180,E1 18096.432,E2 18096.432} C_VEL
LIN {X 0,Y 393.388,Z 404.916,A -85,B 0,C 180,E1 18093.06,E2 18093.06} C_VEL
LIN {X 0,Y 393.563,Z 405.097,A -85,B 0,C 180,E1 18089.709,E2 18089.709} C_VEL
LIN {X 0,Y 393.316,Z 404.882,A -85,B 0,C 180,E1 18086.502,E2 18086.502} C_VEL
LIN {X 0,Y 392.613,Z 404.24,A -85,B 0,C 180,E1 18083.227,E2 18083.227} C_VEL
LIN {X 0,Y 391.621,Z 402.962,A -85,B 0,C 180,E1 18080.151,E2 18080.151} C_VEL
LIN {X 0,Y 390.18,Z 400.306,A -85,B 0,C 180,E1 18076.802,E2 18076.802} C_VEL
LIN {X 0,Y 388.482,Z 399.254,A -85,B 0,C 180,E1 18074.015,E2 18074.015} C_VEL
LIN {X 0,Y 386.185,Z 397.834,A -85,B 0,C 180,E1 18070.879,E2 18070.879} C_VEL
LIN {X 0,Y 384.216,Z 395.508,A -85,B 0,C 180,E1 18068.394,E2 18068.394} C_VEL
LIN {X 0,Y 382.758,Z 392.947,A -85,B 0,C 180,E1 18066.606,E2 18066.606} C_VEL
LIN {X 0,Y 379.378,Z 391.043,A -85,B 0,C 180,E1 18063.286,E2 18063.286} C_VEL
LIN {X 0,Y 377.299,Z 388.586,A -85,B 0,C 180,E1 18061.281,E2 18061.281} C_VEL
LIN {X 0,Y 376.009,Z 386.17,A -85,B 0,C 180,E1 18060.006,E2 18060.006} C_VEL
LIN {X 0,Y 372.14,Z 383.761,A -85,B 0,C 180,E1 18056.856,E2 18056.856} C_VEL
LIN {X 0,Y 370.311,Z 381.215,A -85,B 0,C 180,E1 18055.318,E2 18055.318} C_VEL
LIN {X 0,Y 369.787,Z 379.418,A -85,B 0,C 180,E1 18054.457,E2 18054.457} C_VEL
LIN {X 0,Y 369.703,Z 378.932,A -85,B 0,C 180,E1 18052.65,E2 18052.65} C_VEL
LIN {X 0,Y 369.702,Z 378.936,A -85,B 0,C 180,E1 18052.104,E2 18052.104} C_VEL
LIN {X 0,Y 368.653,Z 379.063,A -85,B 0,C 180,E1 18050.91,E2 18050.91} C_VEL
LIN {X 0,Y 362.15,Z 379.879,A -85,B 0,C 180,E1 18047.452,E2 18047.452} C_VEL
LIN {X 0,Y 361.758,Z 379.923,A -85,B 0,C 180,E1 18046.657,E2 18046.657} C_VEL
LIN {X 0,Y 361.768,Z 379.92,A -85,B 0,C 180,E1 18042.446,E2 18042.446} C_VEL
LIN {X 0,Y 361.782,Z 379.922,A -85,B 0,C 180,E1 18038.236,E2 18038.236} C_VEL
LIN {X 0,Y 361.777,Z 379.923,A -85,B 0,C 180,E1 18033.994,E2 18033.994} C_VEL
LIN {X 0,Y 361.772,Z 379.923,A -85,B 0,C 180,E1 18029.796,E2 18029.796} C_VEL
LIN {X 0,Y 361.763,Z 379.891,A -85,B 0,C 180,E1 18025.707,E2 18025.707} C_VEL
LIN {X 0,Y 361.762,Z 379.911,A -85,B 0,C 180,E1 18021.558,E2 18021.558} C_VEL
LIN {X 0,Y 361.758,Z 379.867,A -85,B 0,C 180,E1 18017.525,E2 18017.525} C_VEL
LIN {X 0,Y 361.761,Z 379.924,A -85,B 0,C 180,E1 18013.416,E2 18013.416} C_VEL
LIN {X 0,Y 361.755,Z 379.863,A -85,B 0,C 180,E1 18009.36,E2 18009.36} C_VEL
LIN {X 0,Y 361.768,Z 379.921,A -85,B 0,C 180,E1 18005.385,E2 18005.385} C_VEL
LIN {X 0,Y 361.755,Z 379.861,A -85,B 0,C 180,E1 18001.26,E2 18001.26} C_VEL
LIN {X 0,Y 361.771,Z 379.921,A -85,B 0,C 180,E1 17997.3,E2 17997.3} C_VEL
LIN {X 0,Y 361.76,Z 379.863,A -85,B 0,C 180,E1 17993.168,E2 17993.168} C_VEL
LIN {X 0,Y 361.77,Z 379.918,A -85,B 0,C 180,E1 17989.161,E2 17989.161} C_VEL
LIN {X 0,Y 361.771,Z 379.867,A -85,B 0,C 180,E1 17985.1,E2 17985.1} C_VEL
LIN {X 0,Y 361.767,Z 379.904,A -85,B 0,C 180,E1 17980.944,E2 17980.944} C_VEL
LIN {X 0,Y 361.767,Z 379.89,A -85,B 0,C 180,E1 17976.886,E2 17976.886} C_VEL
LIN {X 0,Y 361.771,Z 379.877,A -85,B 0,C 180,E1 17972.862,E2 17972.862} C_VEL
LIN {X 0,Y 361.78,Z 379.92,A -85,B 0,C 180,E1 17968.876,E2 17968.876} C_VEL
LIN {X 0,Y 361.77,Z 379.916,A -85,B 0,C 180,E1 17964.71,E2 17964.71} C_VEL
LIN {X 0,Y 361.823,Z 380.217,A -85,B 0,C 180,E1 17962.996,E2 17962.996} C_VEL
LIN {X 0,Y 364.334,Z 387.205,A -85,B 0,C 180,E1 17960.754,E2 17960.754} C_VEL
LIN {X 0,Y 368.514,Z 393.384,A -85,B 0,C 180,E1 17959.773,E2 17959.773} C_VEL
LIN {X 0,Y 378.203,Z 408.641,A -85,B 0,C 180,E1 17957.658,E2 17957.658} C_VEL
LIN {X 0,Y 387.104,Z 423.494,A -85,B 0,C 180,E1 17955.855,E2 17955.855} C_VEL
LIN {X 0,Y 397.066,Z 441.816,A -85,B 0,C 180,E1 17953.952,E2 17953.952} C_VEL
LIN {X 0,Y 401.912,Z 451.938,A -85,B 0,C 180,E1 17953.052,E2 17953.052} C_VEL
LIN {X 0,Y 394.722,Z 646.828,A -85,B 0,C 180,E1 17949.34,E2 17949.34} C_VEL
LIN {X 0,Y 393.081,Z 667.888,A -85,B 0,C 180,E1 17948.743,E2 17948.743} C_VEL
LIN {X 0,Y 390.909,Z 686.805,A -85,B 0,C 180,E1 17947.961,E2 17947.961} C_VEL
LIN {X 0,Y 388.623,Z 703.517,A -85,B 0,C 180,E1 17947.072,E2 17947.072} C_VEL
LIN {X 0,Y 385.578,Z 722.816,A -85,B 0,C 180,E1 17945.784,E2 17945.784} C_VEL
LIN {X 0,Y 382.462,Z 739.638,A -85,B 0,C 180,E1 17944.379,E2 17944.379} C_VEL
LIN {X 0,Y 379.439,Z 754.786,A -85,B 0,C 180,E1 17942.875,E2 17942.875} C_VEL
LIN {X 0,Y 375.922,Z 771.642,A -85,B 0,C 180,E1 17940.885,E2 17940.885} C_VEL
LIN {X 0,Y 372.644,Z 786.29,A -85,B 0,C 180,E1 17938.791,E2 17938.791} C_VEL
LIN {X 0,Y 370.015,Z 798.115,A -85,B 0,C 180,E1 17936.824,E2 17936.824} C_VEL
LIN {X 0,Y 367.181,Z 811.268,A -85,B 0,C 180,E1 17934.278,E2 17934.278} C_VEL
LIN {X 0,Y 364.751,Z 822.861,A -85,B 0,C 180,E1 17931.55,E2 17931.55} C_VEL
LIN {X 0,Y 363.107,Z 831.614,A -85,B 0,C 180,E1 17929.127,E2 17929.127} C_VEL
LIN {X 0,Y 361.673,Z 840.501,A -85,B 0,C 180,E1 17926.213,E2 17926.213} C_VEL
LIN {X 0,Y 360.698,Z 847.91,A -85,B 0,C 180,E1 17923.138,E2 17923.138} C_VEL
LIN {X 0,Y 360.218,Z 853.139,A -85,B 0,C 180,E1 17920.394,E2 17920.394} C_VEL
LIN {X 0,Y 360.01,Z 857.121,A -85,B 0,C 180,E1 17917.661,E2 17917.661} C_VEL
LIN {X 0,Y 359.935,Z 860.359,A -85,B 0,C 180,E1 17914.301,E2 17914.301} C_VEL
LIN {X 0,Y 359.947,Z 861.623,A -85,B 0,C 180,E1 17911.433,E2 17911.433} C_VEL
LIN {X 0,Y 359.952,Z 861.683,A -85,B 0,C 180,E1 17908.886,E2 17908.886} C_VEL
LIN {X 0,Y 359.942,Z 860.716,A -85,B 0,C 180,E1 17906.337,E2 17906.337} C_VEL
LIN {X 0,Y 359.962,Z 858.414,A -85,B 0,C 180,E1 17903.461,E2 17903.461} C_VEL
LIN {X 0,Y 360.17,Z 853.954,A -85,B 0,C 180,E1 17900.089,E2 17900.089} C_VEL
LIN {X 0,Y 360.591,Z 848.917,A -85,B 0,C 180,E1 17897.347,E2 17897.347} C_VEL
LIN {X 0,Y 361.368,Z 842.576,A -85,B 0,C 180,E1 17894.597,E2 17894.597} C_VEL
LIN {X 0,Y 362.832,Z 833.245,A -85,B 0,C 180,E1 17891.358,E2 17891.358} C_VEL
LIN {X 0,Y 364.505,Z 824.104,A -85,B 0,C 180,E1 17888.772,E2 17888.772} C_VEL
LIN {X 0,Y 366.549,Z 814.105,A -85,B 0,C 180,E1 17886.361,E2 17886.361} C_VEL
LIN {X 0,Y 369.509,Z 800.502,A -85,B 0,C 180,E1 17883.6,E2 17883.6} C_VEL
LIN {X 0,Y 372.338,Z 787.649,A -85,B 0,C 180,E1 17881.421,E2 17881.421} C_VEL
LIN {X 0,Y 375.231,Z 774.623,A -85,B 0,C 180,E1 17879.523,E2 17879.523} C_VEL
LIN {X 0,Y 378.877,Z 757.637,A -85,B 0,C 180,E1 17877.429,E2 17877.429} C_VEL
LIN {X 0,Y 382.126,Z 741.363,A -85,B 0,C 180,E1 17875.78,E2 17875.78} C_VEL
LIN {X 0,Y 385.057,Z 725.582,A -85,B 0,C 180,E1 17874.435,E2 17874.435} C_VEL
LIN {X 0,Y 388.341,Z 705.536,A -85,B 0,C 180,E1 17873.046,E2 17873.046} C_VEL
LIN {X 0,Y 390.719,Z 688.293,A -85,B 0,C 180,E1 17872.11,E2 17872.11} C_VEL
LIN {X 0,Y 392.798,Z 670.337,A -85,B 0,C 180,E1 17871.349,E2 17871.349} C_VEL
LIN {X 0,Y 394.669,Z 647.855,A -85,B 0,C 180,E1 17870.683,E2 17870.683} C_VEL
LIN {X 0,Y 397.515,Z 571.864,A -85,B 0,C 180,E1 17869.214,E2 17869.214} C_VEL
LIN {X 0,Y 401.808,Z 451.346,A -85,B 0,C 180,E1 17866.92,E2 17866.92} C_VEL
LIN {X 0,Y 391.602,Z 431.453,A -85,B 0,C 180,E1 17865.016,E2 17865.016} C_VEL
LIN {X 0,Y 382.288,Z 415.304,A -85,B 0,C 180,E1 17863.183,E2 17863.183} C_VEL
LIN {X 0,Y 374.179,Z 402.229,A -85,B 0,C 180,E1 17861.485,E2 17861.485} C_VEL
LIN {X 0,Y 366.936,Z 391.268,A -85,B 0,C 180,E1 17859.874,E2 17859.874} C_VEL
LIN {X 0,Y 364.175,Z 386.774,A -85,B 0,C 180,E1 17859.164,E2 17859.164} C_VEL
LIN {X 0,Y 361.781,Z 379.975,A -85,B 0,C 180,E1 17856.856,E2 17856.856} C_VEL
LIN {X 0,Y 361.772,Z 379.892,A -85,B 0,C 180,E1 17852.805,E2 17852.805} C_VEL
LIN {X 0,Y 361.775,Z 379.878,A -85,B 0,C 180,E1 17848.749,E2 17848.749} C_VEL
LIN {X 0,Y 361.77,Z 379.923,A -85,B 0,C 180,E1 17844.597,E2 17844.597} C_VEL
LIN {X 0,Y 361.767,Z 379.873,A -85,B 0,C 180,E1 17840.555,E2 17840.555} C_VEL
LIN {X 0,Y 361.766,Z 379.9,A -85,B 0,C 180,E1 17836.46,E2 17836.46} C_VEL
LIN {X 0,Y 361.767,Z 379.883,A -85,B 0,C 180,E1 17832.456,E2 17832.456} C_VEL
LIN {X 0,Y 361.766,Z 379.886,A -85,B 0,C 180,E1 17828.341,E2 17828.341} C_VEL
LIN {X 0,Y 361.763,Z 379.892,A -85,B 0,C 180,E1 17824.286,E2 17824.286} C_VEL
LIN {X 0,Y 361.76,Z 379.881,A -85,B 0,C 180,E1 17820.165,E2 17820.165} C_VEL
LIN {X 0,Y 361.757,Z 379.899,A -85,B 0,C 180,E1 17816.045,E2 17816.045} C_VEL
LIN {X 0,Y 361.762,Z 379.877,A -85,B 0,C 180,E1 17812.064,E2 17812.064} C_VEL
LIN {X 0,Y 361.757,Z 379.908,A -85,B 0,C 180,E1 17807.882,E2 17807.882} C_VEL
LIN {X 0,Y 361.764,Z 379.872,A -85,B 0,C 180,E1 17803.964,E2 17803.964} C_VEL
LIN {X 0,Y 361.762,Z 379.921,A -85,B 0,C 180,E1 17799.798,E2 17799.798} C_VEL
LIN {X 0,Y 361.759,Z 379.872,A -85,B 0,C 180,E1 17795.79,E2 17795.79} C_VEL
LIN {X 0,Y 361.761,Z 379.925,A -85,B 0,C 180,E1 17791.626,E2 17791.626} C_VEL
LIN {X 0,Y 361.761,Z 379.924,A -85,B 0,C 180,E1 17787.586,E2 17787.586} C_VEL
LIN {X 0,Y 361.761,Z 379.924,A -85,B 0,C 180,E1 17783.539,E2 17783.539} C_VEL
LIN {X 0,Y 361.761,Z 379.921,A -85,B 0,C 180,E1 17779.468,E2 17779.468} C_VEL
LIN {X 0,Y 361.76,Z 379.921,A -85,B 0,C 180,E1 17775.424,E2 17775.424} C_VEL
LIN {X 0,Y 361.764,Z 379.975,A -85,B 0,C 180,E1 17771.272,E2 17771.272} C_VEL
LIN {X 0,Y 361.966,Z 381.046,A -85,B 0,C 180,E1 17770.268,E2 17770.268} C_VEL
LIN {X 0,Y 363.582,Z 384.113,A -85,B 0,C 180,E1 17768.915,E2 17768.915} C_VEL
LIN {X 0,Y 366.082,Z 386.074,A -85,B 0,C 180,E1 17767.123,E2 17767.123} C_VEL
LIN {X 0,Y 368.196,Z 387.328,A -85,B 0,C 180,E1 17765.597,E2 17765.597} C_VEL
LIN {X 0,Y 369.849,Z 390.357,A -85,B 0,C 180,E1 17764.201,E2 17764.201} C_VEL
LIN {X 0,Y 372.266,Z 392.625,A -85,B 0,C 180,E1 17762.235,E2 17762.235} C_VEL
LIN {X 0,Y 375.027,Z 394.285,A -85,B 0,C 180,E1 17759.968,E2 17759.968} C_VEL
LIN {X 0,Y 376.846,Z 397.515,A -85,B 0,C 180,E1 17758.181,E2 17758.181} C_VEL
LIN {X 0,Y 379.455,Z 399.704,A -85,B 0,C 180,E1 17755.712,E2 17755.712} C_VEL
LIN {X 0,Y 381.895,Z 401.124,A -85,B 0,C 180,E1 17753.25,E2 17753.25} C_VEL
LIN {X 0,Y 383.921,Z 404.525,A -85,B 0,C 180,E1 17750.743,E2 17750.743} C_VEL
LIN {X 0,Y 386.258,Z 406.551,A -85,B 0,C 180,E1 17747.747,E2 17747.747} C_VEL
LIN {X 0,Y 388.51,Z 407.633,A -85,B 0,C 180,E1 17744.456,E2 17744.456} C_VEL
LIN {X 0,Y 389.677,Z 409.142,A -85,B 0,C 180,E1 17742.145,E2 17742.145} C_VEL
LIN {X 0,Y 390.8,Z 411.081,A -85,B 0,C 180,E1 17739.424,E2 17739.424} C_VEL
LIN {X 0,Y 391.782,Z 412.32,A -85,B 0,C 180,E1 17736.3,E2 17736.3} C_VEL
LIN {X 0,Y 392.419,Z 412.865,A -85,B 0,C 180,E1 17732.921,E2 17732.921} C_VEL
LIN {X 0,Y 392.588,Z 413.038,A -85,B 0,C 180,E1 17729.708,E2 17729.708} C_VEL
LIN {X 0,Y 392.34,Z 412.822,A -85,B 0,C 180,E1 17726.494,E2 17726.494} C_VEL
LIN {X 0,Y 391.626,Z 412.181,A -85,B 0,C 180,E1 17723.202,E2 17723.202} C_VEL
LIN {X 0,Y 390.63,Z 410.903,A -85,B 0,C 180,E1 17720.126,E2 17720.126} C_VEL
LIN {X 0,Y 389.185,Z 408.263,A -85,B 0,C 180,E1 17716.783,E2 17716.783} C_VEL
LIN {X 0,Y 387.476,Z 407.186,A -85,B 0,C 180,E1 17713.973,E2 17713.973} C_VEL
LIN {X 0,Y 385.185,Z 405.786,A -85,B 0,C 180,E1 17710.854,E2 17710.854} C_VEL
LIN {X 0,Y 383.093,Z 403.385,A -85,B 0,C 180,E1 17708.247,E2 17708.247} C_VEL
LIN {X 0,Y 381.541,Z 400.723,A -85,B 0,C 180,E1 17706.363,E2 17706.363} C_VEL
LIN {X 0,Y 378.352,Z 399.006,A -85,B 0,C 180,E1 17703.258,E2 17703.258} C_VEL
LIN {X 0,Y 376.069,Z 396.37,A -85,B 0,C 180,E1 17701.062,E2 17701.062} C_VEL
LIN {X 0,Y 374.665,Z 393.879,A -85,B 0,C 180,E1 17699.711,E2 17699.711} C_VEL
LIN {X 0,Y 370.979,Z 391.658,A -85,B 0,C 180,E1 17696.739,E2 17696.739} C_VEL
LIN {X 0,Y 368.873,Z 388.844,A -85,B 0,C 180,E1 17695.001,E2 17695.001} C_VEL
LIN {X 0,Y 367.811,Z 386.932,A -85,B 0,C 180,E1 17694.087,E2 17694.087} C_VEL
LIN {X 0,Y 364.123,Z 384.698,A -85,B 0,C 180,E1 17691.482,E2 17691.482} C_VEL
LIN {X 0,Y 362.377,Z 382.134,A -85,B 0,C 180,E1 17690.15,E2 17690.15} C_VEL
LIN {X 0,Y 361.799,Z 380.35,A -85,B 0,C 180,E1 17689.294,E2 17689.294} C_VEL
LIN {X 0,Y 361.739,Z 379.923,A -85,B 0,C 180,E1 17687.546,E2 17687.546} C_VEL
LIN {X 0,Y 361.758,Z 379.923,A -85,B 0,C 180,E1 17686.657,E2 17686.657} C_VEL
LIN {X 0,Y 360.937,Z 380.027,A -85,B 0,C 180,E1 17685.524,E2 17685.524} C_VEL
LIN {X 0,Y 357.082,Z 380.507,A -85,B 0,C 180,E1 17683.564,E2 17683.564} C_VEL
LIN {X 0,Y 354.147,Z 380.872,A -85,B 0,C 180,E1 17681.814,E2 17681.814} C_VEL
LIN {X 0,Y 353.798,Z 380.913,A -85,B 0,C 180,E1 17681.091,E2 17681.091} C_VEL
LIN {X 0,Y 353.801,Z 380.912,A -85,B 0,C 180,E1 17676.894,E2 17676.894} C_VEL
LIN {X 0,Y 353.802,Z 380.916,A -85,B 0,C 180,E1 17672.85,E2 17672.85} C_VEL
LIN {X 0,Y 353.806,Z 380.914,A -85,B 0,C 180,E1 17668.703,E2 17668.703} C_VEL
LIN {X 0,Y 353.803,Z 380.863,A -85,B 0,C 180,E1 17664.537,E2 17664.537} C_VEL
LIN {X 0,Y 353.806,Z 380.914,A -85,B 0,C 180,E1 17660.504,E2 17660.504} C_VEL
LIN {X 0,Y 353.801,Z 380.857,A -85,B 0,C 180,E1 17656.407,E2 17656.407} C_VEL
LIN {X 0,Y 353.804,Z 380.904,A -85,B 0,C 180,E1 17652.394,E2 17652.394} C_VEL
LIN {X 0,Y 353.802,Z 380.86,A -85,B 0,C 180,E1 17648.279,E2 17648.279} C_VEL
LIN {X 0,Y 353.806,Z 380.893,A -85,B 0,C 180,E1 17644.206,E2 17644.206} C_VEL
LIN {X 0,Y 353.801,Z 380.863,A -85,B 0,C 180,E1 17640.155,E2 17640.155} C_VEL
LIN {X 0,Y 353.805,Z 380.892,A -85,B 0,C 180,E1 17636.104,E2 17636.104} C_VEL
LIN {X 0,Y 353.802,Z 380.867,A -85,B 0,C 180,E1 17632.034,E2 17632.034} C_VEL
LIN {X 0,Y 353.807,Z 380.881,A -85,B 0,C 180,E1 17627.923,E2 17627.923} C_VEL
LIN {X 0,Y 353.806,Z 380.879,A -85,B 0,C 180,E1 17623.907,E2 17623.907} C_VEL
LIN {X 0,Y 353.805,Z 380.868,A -85,B 0,C 180,E1 17619.826,E2 17619.826} C_VEL
LIN {X 0,Y 353.807,Z 380.911,A -85,B 0,C 180,E1 17615.804,E2 17615.804} C_VEL
LIN {X 0,Y 353.809,Z 380.865,A -85,B 0,C 180,E1 17611.65,E2 17611.65} C_VEL
LIN {X 0,Y 353.808,Z 380.888,A -85,B 0,C 180,E1 17607.666,E2 17607.666} C_VEL
LIN {X 0,Y 353.845,Z 381.152,A -85,B 0,C 180,E1 17604.352,E2 17604.352} C_VEL
LIN {X 0,Y 355.874,Z 386.772,A -85,B 0,C 180,E1 17602.453,E2 17602.453} C_VEL
LIN {X 0,Y 359.982,Z 392.597,A -85,B 0,C 180,E1 17601.418,E2 17601.418} C_VEL
LIN {X 0,Y 369.509,Z 407.185,A -85,B 0,C 180,E1 17599.19,E2 17599.19} C_VEL
LIN {X 0,Y 379.275,Z 423.114,A -85,B 0,C 180,E1 17597.088,E2 17597.088} C_VEL
LIN {X 0,Y 389.941,Z 442.411,A -85,B 0,C 180,E1 17594.947,E2 17594.947} C_VEL
LIN {X 0,Y 395.962,Z 454.777,A -85,B 0,C 180,E1 17593.786,E2 17593.786} C_VEL
LIN {X 0,Y 388.548,Z 646.591,A -85,B 0,C 180,E1 17590.09,E2 17590.09} C_VEL
LIN {X 0,Y 386.844,Z 667.697,A -85,B 0,C 180,E1 17589.486,E2 17589.486} C_VEL
LIN {X 0,Y 384.591,Z 686.567,A -85,B 0,C 180,E1 17588.699,E2 17588.699} C_VEL
LIN {X 0,Y 382.23,Z 703.141,A -85,B 0,C 180,E1 17587.81,E2 17587.81} C_VEL
LIN {X 0,Y 379.032,Z 722.576,A -85,B 0,C 180,E1 17586.501,E2 17586.501} C_VEL
LIN {X 0,Y 375.782,Z 739.398,A -85,B 0,C 180,E1 17585.079,E2 17585.079} C_VEL
LIN {X 0,Y 372.71,Z 754.121,A -85,B 0,C 180,E1 17583.601,E2 17583.601} C_VEL
LIN {X 0,Y 369.059,Z 770.83,A -85,B 0,C 180,E1 17581.615,E2 17581.615} C_VEL
LIN {X 0,Y 365.501,Z 785.97,A -85,B 0,C 180,E1 17579.422,E2 17579.422} C_VEL
LIN {X 0,Y 362.703,Z 797.872,A -85,B 0,C 180,E1 17577.41,E2 17577.41} C_VEL
LIN {X 0,Y 359.703,Z 811.025,A -85,B 0,C 180,E1 17574.817,E2 17574.817} C_VEL
LIN {X 0,Y 357.122,Z 822.618,A -85,B 0,C 180,E1 17572.034,E2 17572.034} C_VEL
LIN {X 0,Y 355.313,Z 831.634,A -85,B 0,C 180,E1 17569.481,E2 17569.481} C_VEL
LIN {X 0,Y 353.755,Z 840.717,A -85,B 0,C 180,E1 17566.417,E2 17566.417} C_VEL
LIN {X 0,Y 352.73,Z 848.005,A -85,B 0,C 180,E1 17563.273,E2 17563.273} C_VEL
LIN {X 0,Y 352.246,Z 852.899,A -85,B 0,C 180,E1 17560.632,E2 17560.632} C_VEL
LIN {X 0,Y 352.017,Z 856.883,A -85,B 0,C 180,E1 17557.836,E2 17557.836} C_VEL
LIN {X 0,Y 351.936,Z 860.122,A -85,B 0,C 180,E1 17554.399,E2 17554.399} C_VEL
LIN {X 0,Y 351.95,Z 861.387,A -85,B 0,C 180,E1 17551.465,E2 17551.465} C_VEL
LIN {X 0,Y 351.954,Z 861.446,A -85,B 0,C 180,E1 17548.861,E2 17548.861} C_VEL
LIN {X 0,Y 351.943,Z 860.479,A -85,B 0,C 180,E1 17546.254,E2 17546.254} C_VEL
LIN {X 0,Y 351.967,Z 858.176,A -85,B 0,C 180,E1 17543.312,E2 17543.312} C_VEL
LIN {X 0,Y 352.191,Z 853.714,A -85,B 0,C 180,E1 17539.863,E2 17539.863} C_VEL
LIN {X 0,Y 352.653,Z 848.676,A -85,B 0,C 180,E1 17537.057,E2 17537.057} C_VEL
LIN {X 0,Y 353.492,Z 842.335,A -85,B 0,C 180,E1 17534.245,E2 17534.245} C_VEL
LIN {X 0,Y 355.068,Z 833.003,A -85,B 0,C 180,E1 17530.935,E2 17530.935} C_VEL
LIN {X 0,Y 356.857,Z 823.861,A -85,B 0,C 180,E1 17528.295,E2 17528.295} C_VEL
LIN {X 0,Y 359.032,Z 813.862,A -85,B 0,C 180,E1 17525.835,E2 17525.835} C_VEL
LIN {X 0,Y 362.105,Z 800.551,A -85,B 0,C 180,E1 17523.075,E2 17523.075} C_VEL
LIN {X 0,Y 365.123,Z 787.551,A -85,B 0,C 180,E1 17520.829,E2 17520.829} C_VEL
LIN {X 0,Y 368.11,Z 774.773,A -85,B 0,C 180,E1 17518.932,E2 17518.932} C_VEL
LIN {X 0,Y 371.881,Z 758.108,A -85,B 0,C 180,E1 17516.83,E2 17516.83} C_VEL
LIN {X 0,Y 375.287,Z 741.836,A -85,B 0,C 180,E1 17515.149,E2 17515.149} C_VEL
LIN {X 0,Y 378.139,Z 727.186,A -85,B 0,C 180,E1 17513.869,E2 17513.869} C_VEL
LIN {X 0,Y 381.374,Z 708.909,A -85,B 0,C 180,E1 17512.539,E2 17512.539} C_VEL
LIN {X 0,Y 384.25,Z 689.142,A -85,B 0,C 180,E1 17511.425,E2 17511.425} C_VEL
LIN {X 0,Y 386.341,Z 671.963,A -85,B 0,C 180,E1 17510.676,E2 17510.676} C_VEL
LIN {X 0,Y 388.292,Z 651.316,A -85,B 0,C 180,E1 17510.016,E2 17510.016} C_VEL
LIN {X 0,Y 389.901,Z 614.05,A -85,B 0,C 180,E1 17509.258,E2 17509.258} C_VEL
LIN {X 0,Y 395.855,Z 454.236,A -85,B 0,C 180,E1 17506.186,E2 17506.186} C_VEL
LIN {X 0,Y 385.623,Z 434.357,A -85,B 0,C 180,E1 17504.204,E2 17504.204} C_VEL
LIN {X 0,Y 375.153,Z 416.225,A -85,B 0,C 180,E1 17502.044,E2 17502.044} C_VEL
LIN {X 0,Y 367.148,Z 403.634,A -85,B 0,C 180,E1 17500.28,E2 17500.28} C_VEL
LIN {X 0,Y 363.006,Z 397.299,A -85,B 0,C 180,E1 17499.315,E2 17499.315} C_VEL
LIN {X 0,Y 359.135,Z 391.655,A -85,B 0,C 180,E1 17498.384,E2 17498.384} C_VEL
LIN {X 0,Y 355.581,Z 386.17,A -85,B 0,C 180,E1 17497.405,E2 17497.405} C_VEL
LIN {X 0,Y 353.827,Z 380.991,A -85,B 0,C 180,E1 17495.53,E2 17495.53} C_VEL
LIN {X 0,Y 353.82,Z 380.905,A -85,B 0,C 180,E1 17491.417,E2 17491.417} C_VEL
LIN {X 0,Y 353.824,Z 380.864,A -85,B 0,C 180,E1 17487.25,E2 17487.25} C_VEL
LIN {X 0,Y 353.826,Z 380.878,A -85,B 0,C 180,E1 17483.134,E2 17483.134} C_VEL
LIN {X 0,Y 353.833,Z 380.893,A -85,B 0,C 180,E1 17478.97,E2 17478.97} C_VEL
LIN {X 0,Y 353.845,Z 380.851,A -85,B 0,C 180,E1 17474.739,E2 17474.739} C_VEL
LIN {X 0,Y 353.831,Z 380.912,A -85,B 0,C 180,E1 17470.426,E2 17470.426} C_VEL
LIN {X 0,Y 353.826,Z 380.848,A -85,B 0,C 180,E1 17466.334,E2 17466.334} C_VEL
LIN {X 0,Y 353.82,Z 380.91,A -85,B 0,C 180,E1 17462.112,E2 17462.112} C_VEL
LIN {X 0,Y 353.813,Z 380.849,A -85,B 0,C 180,E1 17458.064,E2 17458.064} C_VEL
LIN {X 0,Y 353.821,Z 380.908,A -85,B 0,C 180,E1 17454.006,E2 17454.006} C_VEL
LIN {X 0,Y 353.813,Z 380.853,A -85,B 0,C 180,E1 17449.917,E2 17449.917} C_VEL
LIN {X 0,Y 353.812,Z 380.904,A -85,B 0,C 180,E1 17445.76,E2 17445.76} C_VEL
LIN {X 0,Y 353.81,Z 380.864,A -85,B 0,C 180,E1 17441.713,E2 17441.713} C_VEL
LIN {X 0,Y 353.82,Z 380.881,A -85,B 0,C 180,E1 17437.758,E2 17437.758} C_VEL
LIN {X 0,Y 353.814,Z 380.897,A -85,B 0,C 180,E1 17433.611,E2 17433.611} C_VEL
LIN {X 0,Y 353.817,Z 380.914,A -85,B 0,C 180,E1 17429.528,E2 17429.528} C_VEL
LIN {X 0,Y 353.81,Z 380.914,A -85,B 0,C 180,E1 17425.399,E2 17425.399} C_VEL
LIN {X 0,Y 353.805,Z 380.911,A -85,B 0,C 180,E1 17421.257,E2 17421.257} C_VEL
LIN {X 0,Y 353.812,Z 380.91,A -85,B 0,C 180,E1 17417.284,E2 17417.284} C_VEL
LIN {X 0,Y 353.878,Z 381.3,A -85,B 0,C 180,E1 17415.397,E2 17415.397} C_VEL
LIN {X 0,Y 354.449,Z 383.224,A -85,B 0,C 180,E1 17414.574,E2 17414.574} C_VEL
LIN {X 0,Y 356.748,Z 386.177,A -85,B 0,C 180,E1 17413.002,E2 17413.002} C_VEL
LIN {X 0,Y 360.19,Z 388.347,A -85,B 0,C 180,E1 17410.717,E2 17410.717} C_VEL
LIN {X 0,Y 362.171,Z 391.762,A -85,B 0,C 180,E1 17409.212,E2 17409.212} C_VEL
LIN {X 0,Y 365.023,Z 394.008,A -85,B 0,C 180,E1 17407.163,E2 17407.163} C_VEL
LIN {X 0,Y 366.921,Z 395.19,A -85,B 0,C 180,E1 17405.804,E2 17405.804} C_VEL
LIN {X 0,Y 368.533,Z 398.08,A -85,B 0,C 180,E1 17404.452,E2 17404.452} C_VEL
LIN {X 0,Y 371.04,Z 400.453,A -85,B 0,C 180,E1 17402.428,E2 17402.428} C_VEL
LIN {X 0,Y 373.765,Z 402.067,A -85,B 0,C 180,E1 17400.192,E2 17400.192} C_VEL
LIN {X 0,Y 375.538,Z 405.204,A -85,B 0,C 180,E1 17398.461,E2 17398.461} C_VEL
LIN {X 0,Y 378.334,Z 407.583,A -85,B 0,C 180,E1 17395.852,E2 17395.852} C_VEL
LIN {X 0,Y 380.799,Z 409.032,A -85,B 0,C 180,E1 17393.357,E2 17393.357} C_VEL
LIN {X 0,Y 382.77,Z 412.312,A -85,B 0,C 180,E1 17390.969,E2 17390.969} C_VEL
LIN {X 0,Y 385.077,Z 414.404,A -85,B 0,C 180,E1 17387.998,E2 17387.998} C_VEL
LIN {X 0,Y 387.424,Z 415.525,A -85,B 0,C 180,E1 17384.622,E2 17384.622} C_VEL
LIN {X 0,Y 388.665,Z 417.09,A -85,B 0,C 180,E1 17382.208,E2 17382.208} C_VEL
LIN {X 0,Y 389.816,Z 419.029,A -85,B 0,C 180,E1 17379.448,E2 17379.448} C_VEL
LIN {X 0,Y 390.805,Z 420.26,A -85,B 0,C 180,E1 17376.316,E2 17376.316} C_VEL
LIN {X 0,Y 391.445,Z 420.805,A -85,B 0,C 180,E1 17372.928,E2 17372.928} C_VEL
LIN {X 0,Y 391.602,Z 420.964,A -85,B 0,C 180,E1 17369.561,E2 17369.561} C_VEL
LIN {X 0,Y 391.331,Z 420.741,A -85,B 0,C 180,E1 17366.338,E2 17366.338} C_VEL
LIN {X 0,Y 390.612,Z 420.086,A -85,B 0,C 180,E1 17363.09,E2 17363.09} C_VEL
LIN {X 0,Y 389.567,Z 418.771,A -85,B 0,C 180,E1 17359.949,E2 17359.949} C_VEL
LIN {X 0,Y 388.091,Z 416.104,A -85,B 0,C 180,E1 17356.593,E2 17356.593} C_VEL
LIN {X 0,Y 386.338,Z 415.067,A -85,B 0,C 180,E1 17353.736,E2 17353.736} C_VEL
LIN {X 0,Y 383.962,Z 413.535,A -85,B 0,C 180,E1 17350.53,E2 17350.53} C_VEL
LIN {X 0,Y 381.907,Z 411.143,A -85,B 0,C 180,E1 17348.014,E2 17348.014} C_VEL
LIN {X 0,Y 380.329,Z 408.519,A -85,B 0,C 180,E1 17346.119,E2 17346.119} C_VEL
LIN {X 0,Y 377.13,Z 406.802,A -85,B 0,C 180,E1 17343.041,E2 17343.041} C_VEL
LIN {X 0,Y 374.785,Z 404.045,A -85,B 0,C 180,E1 17340.778,E2 17340.778} C_VEL
LIN {X 0,Y 373.33,Z 401.59,A -85,B 0,C 180,E1 17339.413,E2 17339.413} C_VEL
LIN {X 0,Y 369.84,Z 399.57,A -85,B 0,C 180,E1 17336.637,E2 17336.637} C_VEL
LIN {X 0,Y 367.466,Z 396.501,A -85,B 0,C 180,E1 17334.697,E2 17334.697} C_VEL
LIN {X 0,Y 366.572,Z 394.751,A -85,B 0,C 180,E1 17333.904,E2 17333.904} C_VEL
LIN {X 0,Y 362.911,Z 392.569,A -85,B 0,C 180,E1 17331.343,E2 17331.343} C_VEL
LIN {X 0,Y 360.915,Z 389.847,A -85,B 0,C 180,E1 17329.857,E2 17329.857} C_VEL
LIN {X 0,Y 359.841,Z 387.949,A -85,B 0,C 180,E1 17329.025,E2 17329.025} C_VEL
LIN {X 0,Y 356.163,Z 385.639,A -85,B 0,C 180,E1 17326.629,E2 17326.629} C_VEL
LIN {X 0,Y 354.26,Z 382.776,A -85,B 0,C 180,E1 17325.264,E2 17325.264} C_VEL
LIN {X 0,Y 353.879,Z 381.304,A -85,B 0,C 180,E1 17324.603,E2 17324.603} C_VEL
LIN {X 0,Y 353.813,Z 380.91,A -85,B 0,C 180,E1 17322.692,E2 17322.692} C_VEL
LIN {X 0,Y 353.798,Z 380.913,A -85,B 0,C 180,E1 17321.091,E2 17321.091} C_VEL
LIN {X 0,Y 352.826,Z 381.038,A -85,B 0,C 180,E1 17319.844,E2 17319.844} C_VEL
LIN {X 0,Y 348.245,Z 381.607,A -85,B 0,C 180,E1 17317.486,E2 17317.486} C_VEL
LIN {X 0,Y 346.015,Z 381.885,A -85,B 0,C 180,E1 17315.86,E2 17315.86} C_VEL
LIN {X 0,Y 345.864,Z 381.904,A -85,B 0,C 180,E1 17315.396,E2 17315.396} C_VEL
LIN {X 0,Y 345.861,Z 381.904,A -85,B 0,C 180,E1 17311.152,E2 17311.152} C_VEL
LIN {X 0,Y 345.86,Z 381.903,A -85,B 0,C 180,E1 17306.982,E2 17306.982} C_VEL
LIN {X 0,Y 345.858,Z 381.86,A -85,B 0,C 180,E1 17302.752,E2 17302.752} C_VEL
LIN {X 0,Y 345.856,Z 381.861,A -85,B 0,C 180,E1 17298.708,E2 17298.708} C_VEL
LIN {X 0,Y 345.86,Z 381.882,A -85,B 0,C 180,E1 17294.558,E2 17294.558} C_VEL
LIN {X 0,Y 345.856,Z 381.846,A -85,B 0,C 180,E1 17290.486,E2 17290.486} C_VEL
LIN {X 0,Y 345.866,Z 381.896,A -85,B 0,C 180,E1 17286.299,E2 17286.299} C_VEL
LIN {X 0,Y 345.863,Z 381.838,A -85,B 0,C 180,E1 17282.146,E2 17282.146} C_VEL
LIN {X 0,Y 345.875,Z 381.899,A -85,B 0,C 180,E1 17278.005,E2 17278.005} C_VEL
LIN {X 0,Y 345.873,Z 381.837,A -85,B 0,C 180,E1 17273.853,E2 17273.853} C_VEL
LIN {X 0,Y 345.887,Z 381.901,A -85,B 0,C 180,E1 17269.669,E2 17269.669} C_VEL
LIN {X 0,Y 345.897,Z 381.838,A -85,B 0,C 180,E1 17265.428,E2 17265.428} C_VEL
LIN {X 0,Y 345.897,Z 381.881,A -85,B 0,C 180,E1 17261.104,E2 17261.104} C_VEL
LIN {X 0,Y 345.885,Z 381.865,A -85,B 0,C 180,E1 17256.844,E2 17256.844} C_VEL
LIN {X 0,Y 345.889,Z 381.852,A -85,B 0,C 180,E1 17252.818,E2 17252.818} C_VEL
LIN {X 0,Y 345.884,Z 381.893,A -85,B 0,C 180,E1 17248.64,E2 17248.64} C_VEL
LIN {X 0,Y 345.9,Z 382.139,A -85,B 0,C 180,E1 17245.784,E2 17245.784} C_VEL
LIN {X 0,Y 347.454,Z 386.314,A -85,B 0,C 180,E1 17244.301,E2 17244.301} C_VEL
LIN {X 0,Y 354.348,Z 396.416,A -85,B 0,C 180,E1 17242.442,E2 17242.442} C_VEL
LIN {X 0,Y 357.399,Z 400.789,A -85,B 0,C 180,E1 17241.677,E2 17241.677} C_VEL
LIN {X 0,Y 362.22,Z 408.097,A -85,B 0,C 180,E1 17240.506,E2 17240.506} C_VEL
LIN {X 0,Y 369.932,Z 420.408,A -85,B 0,C 180,E1 17238.734,E2 17238.734} C_VEL
LIN {X 0,Y 378.675,Z 435.513,A -85,B 0,C 180,E1 17236.848,E2 17236.848} C_VEL
LIN {X 0,Y 387.794,Z 452.838,A -85,B 0,C 180,E1 17234.995,E2 17234.995} C_VEL
LIN {X 0,Y 390.068,Z 457.883,A -85,B 0,C 180,E1 17234.537,E2 17234.537} C_VEL
LIN {X 0,Y 382.444,Z 646.354,A -85,B 0,C 180,E1 17230.864,E2 17230.864} C_VEL
LIN {X 0,Y 380.678,Z 667.459,A -85,B 0,C 180,E1 17230.255,E2 17230.255} C_VEL
LIN {X 0,Y 378.362,Z 686.18,A -85,B 0,C 180,E1 17229.469,E2 17229.469} C_VEL
LIN {X 0,Y 375.934,Z 702.568,A -85,B 0,C 180,E1 17228.585,E2 17228.585} C_VEL
LIN {X 0,Y 372.733,Z 721.401,A -85,B 0,C 180,E1 17227.317,E2 17227.317} C_VEL
LIN {X 0,Y 369.16,Z 739.158,A -85,B 0,C 180,E1 17225.804,E2 17225.804} C_VEL
LIN {X 0,Y 366.017,Z 753.592,A -85,B 0,C 180,E1 17224.339,E2 17224.339} C_VEL
LIN {X 0,Y 362.236,Z 770.081,A -85,B 0,C 180,E1 17222.361,E2 17222.361} C_VEL
LIN {X 0,Y 358.494,Z 785.304,A -85,B 0,C 180,E1 17220.133,E2 17220.133} C_VEL
LIN {X 0,Y 355.434,Z 797.629,A -85,B 0,C 180,E1 17218.019,E2 17218.019} C_VEL
LIN {X 0,Y 352.259,Z 810.782,A -85,B 0,C 180,E1 17215.378,E2 17215.378} C_VEL
LIN {X 0,Y 349.519,Z 822.375,A -85,B 0,C 180,E1 17212.539,E2 17212.539} C_VEL
LIN {X 0,Y 347.635,Z 831.129,A -85,B 0,C 180,E1 17210.014,E2 17210.014} C_VEL
LIN {X 0,Y 345.969,Z 840.124,A -85,B 0,C 180,E1 17206.932,E2 17206.932} C_VEL
LIN {X 0,Y 344.806,Z 847.764,A -85,B 0,C 180,E1 17203.584,E2 17203.584} C_VEL
LIN {X 0,Y 344.256,Z 852.931,A -85,B 0,C 180,E1 17200.712,E2 17200.712} C_VEL
LIN {X 0,Y 344.007,Z 857.273,A -85,B 0,C 180,E1 17197.515,E2 17197.515} C_VEL
LIN {X 0,Y 343.941,Z 860.063,A -85,B 0,C 180,E1 17194.168,E2 17194.168} C_VEL
LIN {X 0,Y 343.955,Z 861.18,A -85,B 0,C 180,E1 17191.333,E2 17191.333} C_VEL
LIN {X 0,Y 343.955,Z 861.18,A -85,B 0,C 180,E1 17188.667,E2 17188.667} C_VEL
LIN {X 0,Y 343.941,Z 860.063,A -85,B 0,C 180,E1 17185.832,E2 17185.832} C_VEL
LIN {X 0,Y 344.011,Z 857.063,A -85,B 0,C 180,E1 17182.317,E2 17182.317} C_VEL
LIN {X 0,Y 344.256,Z 852.931,A -85,B 0,C 180,E1 17179.288,E2 17179.288} C_VEL
LIN {X 0,Y 344.806,Z 847.764,A -85,B 0,C 180,E1 17176.416,E2 17176.416} C_VEL
LIN {X 0,Y 345.969,Z 840.124,A -85,B 0,C 180,E1 17173.068,E2 17173.068} C_VEL
LIN {X 0,Y 347.635,Z 831.129,A -85,B 0,C 180,E1 17169.986,E2 17169.986} C_VEL
LIN {X 0,Y 349.519,Z 822.375,A -85,B 0,C 180,E1 17167.461,E2 17167.461} C_VEL
LIN {X 0,Y 352.259,Z 810.782,A -85,B 0,C 180,E1 17164.622,E2 17164.622} C_VEL
LIN {X 0,Y 355.432,Z 797.629,A -85,B 0,C 180,E1 17161.981,E2 17161.981} C_VEL
LIN {X 0,Y 358.493,Z 785.304,A -85,B 0,C 180,E1 17159.867,E2 17159.867} C_VEL
LIN {X 0,Y 362.398,Z 769.352,A -85,B 0,C 180,E1 17157.547,E2 17157.547} C_VEL
LIN {X 0,Y 366.017,Z 753.592,A -85,B 0,C 180,E1 17155.661,E2 17155.661} C_VEL
LIN {X 0,Y 369.16,Z 739.158,A -85,B 0,C 180,E1 17154.196,E2 17154.196} C_VEL
LIN {X 0,Y 372.734,Z 721.401,A -85,B 0,C 180,E1 17152.683,E2 17152.683} C_VEL
LIN {X 0,Y 375.933,Z 702.568,A -85,B 0,C 180,E1 17151.415,E2 17151.415} C_VEL
LIN {X 0,Y 378.362,Z 686.18,A -85,B 0,C 180,E1 17150.531,E2 17150.531} C_VEL
LIN {X 0,Y 380.846,Z 666.039,A -85,B 0,C 180,E1 17149.693,E2 17149.693} C_VEL
LIN {X 0,Y 382.49,Z 645.532,A -85,B 0,C 180,E1 17149.117,E2 17149.117} C_VEL
LIN {X 0,Y 390.068,Z 457.439,A -85,B 0,C 180,E1 17145.451,E2 17145.451} C_VEL
LIN {X 0,Y 380.314,Z 438.35,A -85,B 0,C 180,E1 17143.488,E2 17143.488} C_VEL
LIN {X 0,Y 370.315,Z 421.023,A -85,B 0,C 180,E1 17141.351,E2 17141.351} C_VEL
LIN {X 0,Y 362.636,Z 408.769,A -85,B 0,C 180,E1 17139.593,E2 17139.593} C_VEL
LIN {X 0,Y 358.971,Z 403.138,A -85,B 0,C 180,E1 17138.71,E2 17138.71} C_VEL
LIN {X 0,Y 355.297,Z 397.713,A -85,B 0,C 180,E1 17137.797,E2 17137.797} C_VEL
LIN {X 0,Y 349.848,Z 389.943,A -85,B 0,C 180,E1 17136.378,E2 17136.378} C_VEL
LIN {X 0,Y 347.231,Z 385.743,A -85,B 0,C 180,E1 17135.573,E2 17135.573} C_VEL
LIN {X 0,Y 345.867,Z 381.924,A -85,B 0,C 180,E1 17134.044,E2 17134.044} C_VEL
LIN {X 0,Y 345.862,Z 381.877,A -85,B 0,C 180,E1 17129.823,E2 17129.823} C_VEL
LIN {X 0,Y 345.87,Z 381.886,A -85,B 0,C 180,E1 17125.589,E2 17125.589} C_VEL
LIN {X 0,Y 345.868,Z 381.846,A -85,B 0,C 180,E1 17121.368,E2 17121.368} C_VEL
LIN {X 0,Y 345.879,Z 381.894,A -85,B 0,C 180,E1 17117.155,E2 17117.155} C_VEL
LIN {X 0,Y 345.878,Z 381.847,A -85,B 0,C 180,E1 17113.038,E2 17113.038} C_VEL
LIN {X 0,Y 345.89,Z 381.872,A -85,B 0,C 180,E1 17108.819,E2 17108.819} C_VEL
LIN {X 0,Y 345.89,Z 381.855,A -85,B 0,C 180,E1 17104.649,E2 17104.649} C_VEL
LIN {X 0,Y 345.904,Z 381.859,A -85,B 0,C 180,E1 17100.504,E2 17100.504} C_VEL
LIN {X 0,Y 345.886,Z 381.866,A -85,B 0,C 180,E1 17096.195,E2 17096.195} C_VEL
LIN {X 0,Y 345.881,Z 381.85,A -85,B 0,C 180,E1 17092.032,E2 17092.032} C_VEL
LIN {X 0,Y 345.875,Z 381.885,A -85,B 0,C 180,E1 17087.826,E2 17087.826} C_VEL
LIN {X 0,Y 345.867,Z 381.845,A -85,B 0,C 180,E1 17083.687,E2 17083.687} C_VEL
LIN {X 0,Y 345.867,Z 381.903,A -85,B 0,C 180,E1 17079.491,E2 17079.491} C_VEL
LIN {X 0,Y 345.862,Z 381.851,A -85,B 0,C 180,E1 17075.409,E2 17075.409} C_VEL
LIN {X 0,Y 345.863,Z 381.903,A -85,B 0,C 180,E1 17071.143,E2 17071.143} C_VEL
LIN {X 0,Y 345.861,Z 381.905,A -85,B 0,C 180,E1 17066.892,E2 17066.892} C_VEL
LIN {X 0,Y 345.862,Z 381.901,A -85,B 0,C 180,E1 17062.633,E2 17062.633} C_VEL
LIN {X 0,Y 345.945,Z 382.197,A -85,B 0,C 180,E1 17059.883,E2 17059.883} C_VEL
LIN {X 0,Y 346.29,Z 383.657,A -85,B 0,C 180,E1 17059.153,E2 17059.153} C_VEL
LIN {X 0,Y 347.863,Z 386.252,A -85,B 0,C 180,E1 17058.109,E2 17058.109} C_VEL
LIN {X 0,Y 350.957,Z 388.403,A -85,B 0,C 180,E1 17056.202,E2 17056.202} C_VEL
LIN {X 0,Y 352.216,Z 389.415,A -85,B 0,C 180,E1 17055.39,E2 17055.39} C_VEL
LIN {X 0,Y 353.949,Z 392.427,A -85,B 0,C 180,E1 17054.165,E2 17054.165} C_VEL
LIN {X 0,Y 356.494,Z 394.694,A -85,B 0,C 180,E1 17052.485,E2 17052.485} C_VEL
LIN {X 0,Y 358.811,Z 396.11,A -85,B 0,C 180,E1 17050.975,E2 17050.975} C_VEL
LIN {X 0,Y 360.775,Z 399.432,A -85,B 0,C 180,E1 17049.497,E2 17049.497} C_VEL
LIN {X 0,Y 363.689,Z 401.796,A -85,B 0,C 180,E1 17047.407,E2 17047.407} C_VEL
LIN {X 0,Y 365.544,Z 402.938,A -85,B 0,C 180,E1 17046.09,E2 17046.09} C_VEL
LIN {X 0,Y 367.2,Z 405.825,A -85,B 0,C 180,E1 17044.686,E2 17044.686} C_VEL
LIN {X 0,Y 369.923,Z 408.348,A -85,B 0,C 180,E1 17042.529,E2 17042.529} C_VEL
LIN {X 0,Y 372.48,Z 409.84,A -85,B 0,C 180,E1 17040.441,E2 17040.441} C_VEL
LIN {X 0,Y 374.436,Z 413.143,A -85,B 0,C 180,E1 17038.553,E2 17038.553} C_VEL
LIN {X 0,Y 377.271,Z 415.495,A -85,B 0,C 180,E1 17035.93,E2 17035.93} C_VEL
LIN {X 0,Y 379.596,Z 416.801,A -85,B 0,C 180,E1 17033.587,E2 17033.587} C_VEL
LIN {X 0,Y 381.613,Z 420.126,A -85,B 0,C 180,E1 17031.161,E2 17031.161} C_VEL
LIN {X 0,Y 383.971,Z 422.287,A -85,B 0,C 180,E1 17028.144,E2 17028.144} C_VEL
LIN {X 0,Y 386.279,Z 423.396,A -85,B 0,C 180,E1 17024.847,E2 17024.847} C_VEL
LIN {X 0,Y 387.557,Z 424.804,A -85,B 0,C 180,E1 17022.516,E2 17022.516} C_VEL
LIN {X 0,Y 388.776,Z 426.903,A -85,B 0,C 180,E1 17019.623,E2 17019.623} C_VEL
LIN {X 0,Y 389.788,Z 428.17,A -85,B 0,C 180,E1 17016.48,E2 17016.48} C_VEL
LIN {X 0,Y 390.459,Z 428.737,A -85,B 0,C 180,E1 17013.082,E2 17013.082} C_VEL
LIN {X 0,Y 390.638,Z 428.92,A -85,B 0,C 180,E1 17009.707,E2 17009.707} C_VEL
LIN {X 0,Y 390.386,Z 428.702,A -85,B 0,C 180,E1 17006.476,E2 17006.476} C_VEL
LIN {X 0,Y 389.628,Z 428.03,A -85,B 0,C 180,E1 17003.073,E2 17003.073} C_VEL
LIN {X 0,Y 388.577,Z 426.714,A -85,B 0,C 180,E1 16999.923,E2 16999.923} C_VEL
LIN {X 0,Y 387.177,Z 424.16,A -85,B 0,C 180,E1 16996.713,E2 16996.713} C_VEL
LIN {X 0,Y 385.56,Z 423.087,A -85,B 0,C 180,E1 16994.045,E2 16994.045} C_VEL
LIN {X 0,Y 383.184,Z 421.687,A -85,B 0,C 180,E1 16990.804,E2 16990.804} C_VEL
LIN {X 0,Y 380.994,Z 419.336,A -85,B 0,C 180,E1 16988.121,E2 16988.121} C_VEL
LIN {X 0,Y 379.277,Z 416.44,A -85,B 0,C 180,E1 16986.048,E2 16986.048} C_VEL
LIN {X 0,Y 376.049,Z 414.716,A -85,B 0,C 180,E1 16982.958,E2 16982.958} C_VEL
LIN {X 0,Y 373.565,Z 411.871,A -85,B 0,C 180,E1 16980.585,E2 16980.585} C_VEL
LIN {X 0,Y 372.167,Z 409.453,A -85,B 0,C 180,E1 16979.264,E2 16979.264} C_VEL
LIN {X 0,Y 368.664,Z 407.443,A -85,B 0,C 180,E1 16976.503,E2 16976.503} C_VEL
LIN {X 0,Y 366.083,Z 404.174,A -85,B 0,C 180,E1 16974.402,E2 16974.402} C_VEL
LIN {X 0,Y 365.122,Z 402.468,A -85,B 0,C 180,E1 16973.602,E2 16973.602} C_VEL
LIN {X 0,Y 361.59,Z 400.334,A -85,B 0,C 180,E1 16971.121,E2 16971.121} C_VEL
LIN {X 0,Y 359.36,Z 397.33,A -85,B 0,C 180,E1 16969.479,E2 16969.479} C_VEL
LIN {X 0,Y 358.411,Z 395.63,A -85,B 0,C 180,E1 16968.733,E2 16968.733} C_VEL
LIN {X 0,Y 354.916,Z 393.53,A -85,B 0,C 180,E1 16966.489,E2 16966.489} C_VEL
LIN {X 0,Y 352.619,Z 390.317,A -85,B 0,C 180,E1 16964.9,E2 16964.9} C_VEL
LIN {X 0,Y 351.656,Z 388.726,A -85,B 0,C 180,E1 16964.235,E2 16964.235} C_VEL
LIN {X 0,Y 348.311,Z 386.695,A -85,B 0,C 180,E1 16962.186,E2 16962.186} C_VEL
LIN {X 0,Y 346.573,Z 384.347,A -85,B 0,C 180,E1 16961.062,E2 16961.062} C_VEL
LIN {X 0,Y 345.983,Z 382.434,A -85,B 0,C 180,E1 16960.328,E2 16960.328} C_VEL
LIN {X 0,Y 345.859,Z 381.901,A -85,B 0,C 180,E1 16959.054,E2 16959.054} C_VEL
LIN {X 0,Y 345.864,Z 381.904,A -85,B 0,C 180,E1 16955.396,E2 16955.396} C_VEL
LIN {X 0,Y 344.874,Z 382.032,A -85,B 0,C 180,E1 16954.12,E2 16954.12} C_VEL
LIN {X 0,Y 340.157,Z 382.618,A -85,B 0,C 180,E1 16951.617,E2 16951.617} C_VEL
LIN {X 0,Y 338.047,Z 382.879,A -85,B 0,C 180,E1 16949.948,E2 16949.948} C_VEL
LIN {X 0,Y 337.94,Z 382.892,A -85,B 0,C 180,E1 16949.568,E2 16949.568} C_VEL
LIN {X 0,Y 337.927,Z 382.848,A -85,B 0,C 180,E1 16945.396,E2 16945.396} C_VEL
LIN {X 0,Y 337.926,Z 382.886,A -85,B 0,C 180,E1 16941.151,E2 16941.151} C_VEL
LIN {X 0,Y 337.915,Z 382.83,A -85,B 0,C 180,E1 16936.847,E2 16936.847} C_VEL
LIN {X 0,Y 337.921,Z 382.886,A -85,B 0,C 180,E1 16932.639,E2 16932.639} C_VEL
LIN {X 0,Y 337.922,Z 382.833,A -85,B 0,C 180,E1 16928.328,E2 16928.328} C_VEL
LIN {X 0,Y 337.928,Z 382.868,A -85,B 0,C 180,E1 16924.234,E2 16924.234} C_VEL
LIN {X 0,Y 337.931,Z 382.838,A -85,B 0,C 180,E1 16919.993,E2 16919.993} C_VEL
LIN {X 0,Y 337.943,Z 382.852,A -85,B 0,C 180,E1 16915.751,E2 16915.751} C_VEL
LIN {X 0,Y 337.958,Z 382.848,A -85,B 0,C 180,E1 16911.486,E2 16911.486} C_VEL
LIN {X 0,Y 337.95,Z 382.835,A -85,B 0,C 180,E1 16907.173,E2 16907.173} C_VEL
LIN {X 0,Y 337.946,Z 382.879,A -85,B 0,C 180,E1 16902.962,E2 16902.962} C_VEL
LIN {X 0,Y 337.936,Z 382.832,A -85,B 0,C 180,E1 16898.744,E2 16898.744} C_VEL
LIN {X 0,Y 337.933,Z 382.874,A -85,B 0,C 180,E1 16894.474,E2 16894.474} C_VEL
LIN {X 0,Y 337.923,Z 382.864,A -85,B 0,C 180,E1 16890.187,E2 16890.187} C_VEL
LIN {X 0,Y 337.964,Z 383.018,A -85,B 0,C 180,E1 16887.416,E2 16887.416} C_VEL
LIN {X 0,Y 338.834,Z 385.678,A -85,B 0,C 180,E1 16886.401,E2 16886.401} C_VEL
LIN {X 0,Y 343.362,Z 391.813,A -85,B 0,C 180,E1 16885.039,E2 16885.039} C_VEL
LIN {X 0,Y 350.701,Z 402.613,A -85,B 0,C 180,E1 16883.012,E2 16883.012} C_VEL
LIN {X 0,Y 354.37,Z 408.066,A -85,B 0,C 180,E1 16882.062,E2 16882.062} C_VEL
LIN {X 0,Y 358.658,Z 414.651,A -85,B 0,C 180,E1 16880.993,E2 16880.993} C_VEL
LIN {X 0,Y 367.749,Z 429.381,A -85,B 0,C 180,E1 16878.86,E2 16878.86} C_VEL
LIN {X 0,Y 377.775,Z 447.498,A -85,B 0,C 180,E1 16876.668,E2 16876.668} C_VEL
LIN {X 0,Y 384.251,Z 460.756,A -85,B 0,C 180,E1 16875.316,E2 16875.316} C_VEL
LIN {X 0,Y 376.406,Z 646.219,A -85,B 0,C 180,E1 16871.661,E2 16871.661} C_VEL
LIN {X 0,Y 374.557,Z 667.437,A -85,B 0,C 180,E1 16871.04,E2 16871.04} C_VEL
LIN {X 0,Y 372.161,Z 686.089,A -85,B 0,C 180,E1 16870.249,E2 16870.249} C_VEL
LIN {X 0,Y 369.659,Z 702.329,A -85,B 0,C 180,E1 16869.365,E2 16869.365} C_VEL
LIN {X 0,Y 366.322,Z 721.162,A -85,B 0,C 180,E1 16868.086,E2 16868.086} C_VEL
LIN {X 0,Y 362.599,Z 738.917,A -85,B 0,C 180,E1 16866.555,E2 16866.555} C_VEL
LIN {X 0,Y 359.321,Z 753.35,A -85,B 0,C 180,E1 16865.071,E2 16865.071} C_VEL
LIN {X 0,Y 355.529,Z 769.111,A -85,B 0,C 180,E1 16863.16,E2 16863.16} C_VEL
LIN {X 0,Y 351.564,Z 784.561,A -85,B 0,C 180,E1 16860.886,E2 16860.886} C_VEL
LIN {X 0,Y 348.208,Z 797.387,A -85,B 0,C 180,E1 16858.654,E2 16858.654} C_VEL
LIN {X 0,Y 344.85,Z 810.539,A -85,B 0,C 180,E1 16855.963,E2 16855.963} C_VEL
LIN {X 0,Y 341.941,Z 822.133,A -85,B 0,C 180,E1 16853.067,E2 16853.067} C_VEL
LIN {X 0,Y 339.931,Z 830.886,A -85,B 0,C 180,E1 16850.488,E2 16850.488} C_VEL
LIN {X 0,Y 338.163,Z 839.775,A -85,B 0,C 180,E1 16847.375,E2 16847.375} C_VEL
LIN {X 0,Y 336.897,Z 847.463,A -85,B 0,C 180,E1 16843.941,E2 16843.941} C_VEL
LIN {X 0,Y 336.317,Z 852.42,A -85,B 0,C 180,E1 16841.142,E2 16841.142} C_VEL
LIN {X 0,Y 336.029,Z 856.406,A -85,B 0,C 180,E1 16838.211,E2 16838.211} C_VEL
LIN {X 0,Y 335.941,Z 859.647,A -85,B 0,C 180,E1 16834.609,E2 16834.609} C_VEL
LIN {X 0,Y 335.956,Z 860.914,A -85,B 0,C 180,E1 16831.535,E2 16831.535} C_VEL
LIN {X 0,Y 335.96,Z 860.974,A -85,B 0,C 180,E1 16828.806,E2 16828.806} C_VEL
LIN {X 0,Y 335.946,Z 860.005,A -85,B 0,C 180,E1 16826.075,E2 16826.075} C_VEL
LIN {X 0,Y 335.984,Z 857.701,A -85,B 0,C 180,E1 16822.992,E2 16822.992} C_VEL
LIN {X 0,Y 336.244,Z 853.235,A -85,B 0,C 180,E1 16819.376,E2 16819.376} C_VEL
LIN {X 0,Y 336.797,Z 848.195,A -85,B 0,C 180,E1 16816.437,E2 16816.437} C_VEL
LIN {X 0,Y 337.777,Z 841.851,A -85,B 0,C 180,E1 16813.491,E2 16813.491} C_VEL
LIN {X 0,Y 339.682,Z 832.079,A -85,B 0,C 180,E1 16809.891,E2 16809.891} C_VEL
LIN {X 0,Y 341.728,Z 823.023,A -85,B 0,C 180,E1 16807.178,E2 16807.178} C_VEL
LIN {X 0,Y 344.279,Z 812.671,A -85,B 0,C 180,E1 16804.544,E2 16804.544} C_VEL
LIN {X 0,Y 347.873,Z 798.693,A -85,B 0,C 180,E1 16801.59,E2 16801.59} C_VEL
LIN {X 0,Y 351.166,Z 786.064,A -85,B 0,C 180,E1 16799.36,E2 16799.36} C_VEL
LIN {X 0,Y 354.782,Z 772.041,A -85,B 0,C 180,E1 16797.243,E2 16797.243} C_VEL
LIN {X 0,Y 358.921,Z 755.066,A -85,B 0,C 180,E1 16795.118,E2 16795.118} C_VEL
LIN {X 0,Y 362.374,Z 739.942,A -85,B 0,C 180,E1 16793.543,E2 16793.543} C_VEL
LIN {X 0,Y 365.743,Z 723.941,A -85,B 0,C 180,E1 16792.142,E2 16792.142} C_VEL
LIN {X 0,Y 369.456,Z 703.574,A -85,B 0,C 180,E1 16790.709,E2 16790.709} C_VEL
LIN {X 0,Y 372.052,Z 686.834,A -85,B 0,C 180,E1 16789.787,E2 16789.787} C_VEL
LIN {X 0,Y 374.401,Z 668.655,A -85,B 0,C 180,E1 16789.006,E2 16789.006} C_VEL
LIN {X 0,Y 376.369,Z 646.836,A -85,B 0,C 180,E1 16788.353,E2 16788.353} C_VEL
LIN {X 0,Y 380.316,Z 553.903,A -85,B 0,C 180,E1 16786.501,E2 16786.501} C_VEL
LIN {X 0,Y 384.144,Z 460.236,A -85,B 0,C 180,E1 16784.654,E2 16784.654} C_VEL
LIN {X 0,Y 375.057,Z 442.484,A -85,B 0,C 180,E1 16782.755,E2 16782.755} C_VEL
LIN {X 0,Y 366.061,Z 426.639,A -85,B 0,C 180,E1 16780.759,E2 16780.759} C_VEL
LIN {X 0,Y 356.488,Z 411.063,A -85,B 0,C 180,E1 16778.464,E2 16778.464} C_VEL
LIN {X 0,Y 346.927,Z 396.975,A -85,B 0,C 180,E1 16775.966,E2 16775.966} C_VEL
LIN {X 0,Y 342.584,Z 390.988,A -85,B 0,C 180,E1 16774.746,E2 16774.746} C_VEL
LIN {X 0,Y 338.556,Z 385.093,A -85,B 0,C 180,E1 16773.427,E2 16773.427} C_VEL
LIN {X 0,Y 337.952,Z 382.964,A -85,B 0,C 180,E1 16772.524,E2 16772.524} C_VEL
LIN {X 0,Y 337.928,Z 382.84,A -85,B 0,C 180,E1 16768.262,E2 16768.262} C_VEL
LIN {X 0,Y 337.924,Z 382.876,A -85,B 0,C 180,E1 16763.92,E2 16763.92} C_VEL
LIN {X 0,Y 337.925,Z 382.854,A -85,B 0,C 180,E1 16759.539,E2 16759.539} C_VEL
LIN {X 0,Y 337.927,Z 382.836,A -85,B 0,C 180,E1 16755.304,E2 16755.304} C_VEL
LIN {X 0,Y 337.938,Z 382.882,A -85,B 0,C 180,E1 16751.095,E2 16751.095} C_VEL
LIN {X 0,Y 337.944,Z 382.823,A -85,B 0,C 180,E1 16746.804,E2 16746.804} C_VEL
LIN {X 0,Y 337.957,Z 382.889,A -85,B 0,C 180,E1 16742.551,E2 16742.551} C_VEL
LIN {X 0,Y 337.949,Z 382.82,A -85,B 0,C 180,E1 16738.312,E2 16738.312} C_VEL
LIN {X 0,Y 337.947,Z 382.886,A -85,B 0,C 180,E1 16734.064,E2 16734.064} C_VEL
LIN {X 0,Y 337.936,Z 382.826,A -85,B 0,C 180,E1 16729.955,E2 16729.955} C_VEL
LIN {X 0,Y 337.936,Z 382.878,A -85,B 0,C 180,E1 16725.793,E2 16725.793} C_VEL
LIN {X 0,Y 337.924,Z 382.842,A -85,B 0,C 180,E1 16721.552,E2 16721.552} C_VEL
LIN {X 0,Y 337.922,Z 382.849,A -85,B 0,C 180,E1 16717.388,E2 16717.388} C_VEL
LIN {X 0,Y 337.922,Z 382.889,A -85,B 0,C 180,E1 16713.093,E2 16713.093} C_VEL
LIN {X 0,Y 337.924,Z 382.892,A -85,B 0,C 180,E1 16708.768,E2 16708.768} C_VEL
LIN {X 0,Y 337.936,Z 382.94,A -85,B 0,C 180,E1 16704.451,E2 16704.451} C_VEL
LIN {X 0,Y 338.131,Z 383.861,A -85,B 0,C 180,E1 16703.65,E2 16703.65} C_VEL
LIN {X 0,Y 339.702,Z 387,A -85,B 0,C 180,E1 16702.476,E2 16702.476} C_VEL
LIN {X 0,Y 342.364,Z 389.097,A -85,B 0,C 180,E1 16700.902,E2 16700.902} C_VEL
LIN {X 0,Y 344.264,Z 390.363,A -85,B 0,C 180,E1 16699.802,E2 16699.802} C_VEL
LIN {X 0,Y 346.04,Z 393.584,A -85,B 0,C 180,E1 16698.585,E2 16698.585} C_VEL
LIN {X 0,Y 349.255,Z 396.067,A -85,B 0,C 180,E1 16696.614,E2 16696.614} C_VEL
LIN {X 0,Y 350.556,Z 396.899,A -85,B 0,C 180,E1 16695.798,E2 16695.798} C_VEL
LIN {X 0,Y 352.71,Z 400.354,A -85,B 0,C 180,E1 16694.307,E2 16694.307} C_VEL
LIN {X 0,Y 355.413,Z 402.628,A -85,B 0,C 180,E1 16692.533,E2 16692.533} C_VEL
LIN {X 0,Y 357.356,Z 403.842,A -85,B 0,C 180,E1 16691.272,E2 16691.272} C_VEL
LIN {X 0,Y 359.397,Z 407.177,A -85,B 0,C 180,E1 16689.731,E2 16689.731} C_VEL
LIN {X 0,Y 362.482,Z 409.649,A -85,B 0,C 180,E1 16687.559,E2 16687.559} C_VEL
LIN {X 0,Y 364.114,Z 410.658,A -85,B 0,C 180,E1 16686.379,E2 16686.379} C_VEL
LIN {X 0,Y 366.011,Z 413.73,A -85,B 0,C 180,E1 16684.815,E2 16684.815} C_VEL
LIN {X 0,Y 368.882,Z 416.289,A -85,B 0,C 180,E1 16682.564,E2 16682.564} C_VEL
LIN {X 0,Y 371.25,Z 417.711,A -85,B 0,C 180,E1 16680.642,E2 16680.642} C_VEL
LIN {X 0,Y 373.336,Z 421.075,A -85,B 0,C 180,E1 16678.645,E2 16678.645} C_VEL
LIN {X 0,Y 376.193,Z 423.405,A -85,B 0,C 180,E1 16676.01,E2 16676.01} C_VEL
LIN {X 0,Y 378.576,Z 424.822,A -85,B 0,C 180,E1 16673.611,E2 16673.611} C_VEL
LIN {X 0,Y 380.38,Z 427.861,A -85,B 0,C 180,E1 16671.43,E2 16671.43} C_VEL
LIN {X 0,Y 382.762,Z 430.1,A -85,B 0,C 180,E1 16668.425,E2 16668.425} C_VEL
LIN {X 0,Y 385.054,Z 431.223,A -85,B 0,C 180,E1 16665.204,E2 16665.204} C_VEL
LIN {X 0,Y 386.47,Z 432.543,A -85,B 0,C 180,E1 16662.793,E2 16662.793} C_VEL
LIN {X 0,Y 387.733,Z 434.783,A -85,B 0,C 180,E1 16659.799,E2 16659.799} C_VEL
LIN {X 0,Y 388.804,Z 436.109,A -85,B 0,C 180,E1 16656.497,E2 16656.497} C_VEL
LIN {X 0,Y 389.481,Z 436.677,A -85,B 0,C 180,E1 16653.09,E2 16653.09} C_VEL
LIN {X 0,Y 389.663,Z 436.861,A -85,B 0,C 180,E1 16649.706,E2 16649.706} C_VEL
LIN {X 0,Y 389.41,Z 436.642,A -85,B 0,C 180,E1 16646.467,E2 16646.467} C_VEL
LIN {X 0,Y 388.645,Z 435.973,A -85,B 0,C 180,E1 16643.055,E2 16643.055} C_VEL
LIN {X 0,Y 387.586,Z 434.655,A -85,B 0,C 180,E1 16639.897,E2 16639.897} C_VEL
LIN {X 0,Y 386.173,Z 432.111,A -85,B 0,C 180,E1 16636.678,E2 16636.678} C_VEL
LIN {X 0,Y 384.554,Z 431.019,A -85,B 0,C 180,E1 16634.002,E2 16634.002} C_VEL
LIN {X 0,Y 382.161,Z 429.62,A -85,B 0,C 180,E1 16630.753,E2 16630.753} C_VEL
LIN {X 0,Y 379.946,Z 427.299,A -85,B 0,C 180,E1 16628.058,E2 16628.058} C_VEL
LIN {X 0,Y 378.076,Z 424.29,A -85,B 0,C 180,E1 16625.812,E2 16625.812} C_VEL
LIN {X 0,Y 374.969,Z 422.629,A -85,B 0,C 180,E1 16622.873,E2 16622.873} C_VEL
LIN {X 0,Y 372.372,Z 419.763,A -85,B 0,C 180,E1 16620.435,E2 16620.435} C_VEL
LIN {X 0,Y 370.861,Z 417.261,A -85,B 0,C 180,E1 16619,E2 16619} C_VEL
LIN {X 0,Y 367.377,Z 415.208,A -85,B 0,C 180,E1 16616.276,E2 16616.276} C_VEL
LIN {X 0,Y 364.64,Z 411.708,A -85,B 0,C 180,E1 16614.045,E2 16614.045} C_VEL
LIN {X 0,Y 363.765,Z 410.271,A -85,B 0,C 180,E1 16613.362,E2 16613.362} C_VEL
LIN {X 0,Y 360.226,Z 408.05,A -85,B 0,C 180,E1 16610.861,E2 16610.861} C_VEL
LIN {X 0,Y 357.821,Z 404.815,A -85,B 0,C 180,E1 16609.097,E2 16609.097} C_VEL
LIN {X 0,Y 356.845,Z 403.311,A -85,B 0,C 180,E1 16608.391,E2 16608.391} C_VEL
LIN {X 0,Y 353.53,Z 401.276,A -85,B 0,C 180,E1 16606.256,E2 16606.256} C_VEL
LIN {X 0,Y 351.07,Z 397.973,A -85,B 0,C 180,E1 16604.577,E2 16604.577} C_VEL
LIN {X 0,Y 350.15,Z 396.44,A -85,B 0,C 180,E1 16603.925,E2 16603.925} C_VEL
LIN {X 0,Y 346.783,Z 394.311,A -85,B 0,C 180,E1 16601.859,E2 16601.859} C_VEL
LIN {X 0,Y 344.81,Z 391.652,A -85,B 0,C 180,E1 16600.603,E2 16600.603} C_VEL
LIN {X 0,Y 343.758,Z 389.769,A -85,B 0,C 180,E1 16599.879,E2 16599.879} C_VEL
LIN {X 0,Y 340.144,Z 387.477,A -85,B 0,C 180,E1 16597.786,E2 16597.786} C_VEL
LIN {X 0,Y 338.299,Z 384.466,A -85,B 0,C 180,E1 16596.542,E2 16596.542} C_VEL
LIN {X 0,Y 338.015,Z 383.288,A -85,B 0,C 180,E1 16596.049,E2 16596.049} C_VEL
LIN {X 0,Y 337.955,Z 382.89,A -85,B 0,C 180,E1 16594.191,E2 16594.191} C_VEL
LIN {X 0,Y 337.964,Z 382.888,A -85,B 0,C 180,E1 16589.91,E2 16589.91} C_VEL
LIN {X 0,Y 337.94,Z 382.892,A -85,B 0,C 180,E1 16589.568,E2 16589.568} C_VEL
LIN {X 0,Y 336.927,Z 383.018,A -85,B 0,C 180,E1 16588.262,E2 16588.262} C_VEL
LIN {X 0,Y 330.375,Z 383.778,A -85,B 0,C 180,E1 16584.376,E2 16584.376} C_VEL
LIN {X 0,Y 330,Z 383.822,A -85,B 0,C 180,E1 16583.601,E2 16583.601} C_VEL
LIN {X 0,Y 329.999,Z 383.851,A -85,B 0,C 180,E1 16579.459,E2 16579.459} C_VEL
LIN {X 0,Y 329.981,Z 383.84,A -85,B 0,C 180,E1 16575.096,E2 16575.096} C_VEL
LIN {X 0,Y 329.981,Z 383.827,A -85,B 0,C 180,E1 16570.977,E2 16570.977} C_VEL
LIN {X 0,Y 329.98,Z 383.862,A -85,B 0,C 180,E1 16566.604,E2 16566.604} C_VEL
LIN {X 0,Y 329.981,Z 383.813,A -85,B 0,C 180,E1 16562.25,E2 16562.25} C_VEL
LIN {X 0,Y 329.993,Z 383.877,A -85,B 0,C 180,E1 16558.083,E2 16558.083} C_VEL
LIN {X 0,Y 330.002,Z 383.809,A -85,B 0,C 180,E1 16553.731,E2 16553.731} C_VEL
LIN {X 0,Y 330.016,Z 383.877,A -85,B 0,C 180,E1 16549.519,E2 16549.519} C_VEL
LIN {X 0,Y 330.014,Z 383.814,A -85,B 0,C 180,E1 16545.118,E2 16545.118} C_VEL
LIN {X 0,Y 330.005,Z 383.849,A -85,B 0,C 180,E1 16540.893,E2 16540.893} C_VEL
LIN {X 0,Y 329.993,Z 383.846,A -85,B 0,C 180,E1 16536.608,E2 16536.608} C_VEL
LIN {X 0,Y 329.988,Z 383.827,A -85,B 0,C 180,E1 16532.375,E2 16532.375} C_VEL
LIN {X 0,Y 330.066,Z 384.129,A -85,B 0,C 180,E1 16529.065,E2 16529.065} C_VEL
LIN {X 0,Y 330.431,Z 385.628,A -85,B 0,C 180,E1 16528.631,E2 16528.631} C_VEL
LIN {X 0,Y 332.317,Z 388.575,A -85,B 0,C 180,E1 16527.969,E2 16527.969} C_VEL
LIN {X 0,Y 335.589,Z 392.235,A -85,B 0,C 180,E1 16526.953,E2 16526.953} C_VEL
LIN {X 0,Y 341.346,Z 400.421,A -85,B 0,C 180,E1 16525.212,E2 16525.212} C_VEL
LIN {X 0,Y 346.703,Z 408.202,A -85,B 0,C 180,E1 16523.701,E2 16523.701} C_VEL
LIN {X 0,Y 354.05,Z 419.395,A -85,B 0,C 180,E1 16521.764,E2 16521.764} C_VEL
LIN {X 0,Y 363.627,Z 435.215,A -85,B 0,C 180,E1 16519.43,E2 16519.43} C_VEL
LIN {X 0,Y 373.337,Z 453.059,A -85,B 0,C 180,E1 16517.236,E2 16517.236} C_VEL
LIN {X 0,Y 378.499,Z 463.801,A -85,B 0,C 180,E1 16516.116,E2 16516.116} C_VEL
LIN {X 0,Y 370.448,Z 645.982,A -85,B 0,C 180,E1 16512.487,E2 16512.487} C_VEL
LIN {X 0,Y 368.549,Z 667.099,A -85,B 0,C 180,E1 16511.864,E2 16511.864} C_VEL
LIN {X 0,Y 366.076,Z 685.705,A -85,B 0,C 180,E1 16511.071,E2 16511.071} C_VEL
LIN {X 0,Y 363.456,Z 702.09,A -85,B 0,C 180,E1 16510.172,E2 16510.172} C_VEL
LIN {X 0,Y 359.98,Z 720.922,A -85,B 0,C 180,E1 16508.881,E2 16508.881} C_VEL
LIN {X 0,Y 356.104,Z 738.677,A -85,B 0,C 180,E1 16507.334,E2 16507.334} C_VEL
LIN {X 0,Y 352.512,Z 753.823,A -85,B 0,C 180,E1 16505.752,E2 16505.752} C_VEL
LIN {X 0,Y 348.247,Z 770.675,A -85,B 0,C 180,E1 16503.649,E2 16503.649} C_VEL
LIN {X 0,Y 344.278,Z 785.321,A -85,B 0,C 180,E1 16501.419,E2 16501.419} C_VEL
LIN {X 0,Y 341.03,Z 797.144,A -85,B 0,C 180,E1 16499.315,E2 16499.315} C_VEL
LIN {X 0,Y 337.479,Z 810.296,A -85,B 0,C 180,E1 16496.574,E2 16496.574} C_VEL
LIN {X 0,Y 334.392,Z 821.89,A -85,B 0,C 180,E1 16493.619,E2 16493.619} C_VEL
LIN {X 0,Y 332.252,Z 830.643,A -85,B 0,C 180,E1 16490.984,E2 16490.984} C_VEL
LIN {X 0,Y 330.354,Z 839.533,A -85,B 0,C 180,E1 16487.799,E2 16487.799} C_VEL
LIN {X 0,Y 329.031,Z 846.946,A -85,B 0,C 180,E1 16484.429,E2 16484.429} C_VEL
LIN {X 0,Y 328.358,Z 852.18,A -85,B 0,C 180,E1 16481.415,E2 16481.415} C_VEL
LIN {X 0,Y 328.04,Z 856.167,A -85,B 0,C 180,E1 16478.412,E2 16478.412} C_VEL
LIN {X 0,Y 327.945,Z 859.321,A -85,B 0,C 180,E1 16474.897,E2 16474.897} C_VEL
LIN {X 0,Y 327.958,Z 860.648,A -85,B 0,C 180,E1 16471.747,E2 16471.747} C_VEL
LIN {X 0,Y 327.965,Z 860.767,A -85,B 0,C 180,E1 16468.952,E2 16468.952} C_VEL
LIN {X 0,Y 327.948,Z 859.857,A -85,B 0,C 180,E1 16466.154,E2 16466.154} C_VEL
LIN {X 0,Y 327.975,Z 857.761,A -85,B 0,C 180,E1 16463.172,E2 16463.172} C_VEL
LIN {X 0,Y 328.211,Z 853.811,A -85,B 0,C 180,E1 16459.646,E2 16459.646} C_VEL
LIN {X 0,Y 328.833,Z 848.29,A -85,B 0,C 180,E1 16456.281,E2 16456.281} C_VEL
LIN {X 0,Y 329.835,Z 842.162,A -85,B 0,C 180,E1 16453.331,E2 16453.331} C_VEL
LIN {X 0,Y 331.662,Z 833.363,A -85,B 0,C 180,E1 16449.9,E2 16449.9} C_VEL
LIN {X 0,Y 334.034,Z 823.308,A -85,B 0,C 180,E1 16446.78,E2 16446.78} C_VEL
LIN {X 0,Y 336.627,Z 813.324,A -85,B 0,C 180,E1 16444.164,E2 16444.164} C_VEL
LIN {X 0,Y 340.313,Z 799.823,A -85,B 0,C 180,E1 16441.195,E2 16441.195} C_VEL
LIN {X 0,Y 343.867,Z 786.824,A -85,B 0,C 180,E1 16438.832,E2 16438.832} C_VEL
LIN {X 0,Y 347.318,Z 774.048,A -85,B 0,C 180,E1 16436.842,E2 16436.842} C_VEL
LIN {X 0,Y 351.659,Z 757.385,A -85,B 0,C 180,E1 16434.649,E2 16434.649} C_VEL
LIN {X 0,Y 355.551,Z 741.1,A -85,B 0,C 180,E1 16432.902,E2 16432.902} C_VEL
LIN {X 0,Y 358.786,Z 726.468,A -85,B 0,C 180,E1 16431.579,E2 16431.579} C_VEL
LIN {X 0,Y 362.422,Z 708.192,A -85,B 0,C 180,E1 16430.206,E2 16430.206} C_VEL
LIN {X 0,Y 365.608,Z 688.829,A -85,B 0,C 180,E1 16429.083,E2 16429.083} C_VEL
LIN {X 0,Y 367.953,Z 671.678,A -85,B 0,C 180,E1 16428.314,E2 16428.314} C_VEL
LIN {X 0,Y 370.12,Z 651.25,A -85,B 0,C 180,E1 16427.637,E2 16427.637} C_VEL
LIN {X 0,Y 371.861,Z 616.397,A -85,B 0,C 180,E1 16426.897,E2 16426.897} C_VEL
LIN {X 0,Y 378.376,Z 463.235,A -85,B 0,C 180,E1 16423.85,E2 16423.85} C_VEL
LIN {X 0,Y 369.652,Z 446.154,A -85,B 0,C 180,E1 16421.952,E2 16421.952} C_VEL
LIN {X 0,Y 359.727,Z 428.523,A -85,B 0,C 180,E1 16419.64,E2 16419.64} C_VEL
LIN {X 0,Y 351.434,Z 415.348,A -85,B 0,C 180,E1 16417.563,E2 16417.563} C_VEL
LIN {X 0,Y 343.503,Z 403.395,A -85,B 0,C 180,E1 16415.403,E2 16415.403} C_VEL
LIN {X 0,Y 339.105,Z 397.278,A -85,B 0,C 180,E1 16414.128,E2 16414.128} C_VEL
LIN {X 0,Y 333.425,Z 389.519,A -85,B 0,C 180,E1 16412.369,E2 16412.369} C_VEL
LIN {X 0,Y 330.951,Z 386.781,A -85,B 0,C 180,E1 16411.582,E2 16411.582} C_VEL
LIN {X 0,Y 330.116,Z 384.449,A -85,B 0,C 180,E1 16411.098,E2 16411.098} C_VEL
LIN {X 0,Y 329.993,Z 383.863,A -85,B 0,C 180,E1 16410.287,E2 16410.287} C_VEL
LIN {X 0,Y 329.987,Z 383.847,A -85,B 0,C 180,E1 16406.069,E2 16406.069} C_VEL
LIN {X 0,Y 329.982,Z 383.822,A -85,B 0,C 180,E1 16401.701,E2 16401.701} C_VEL
LIN {X 0,Y 329.992,Z 383.876,A -85,B 0,C 180,E1 16397.369,E2 16397.369} C_VEL
LIN {X 0,Y 329.993,Z 383.82,A -85,B 0,C 180,E1 16393.142,E2 16393.142} C_VEL
LIN {X 0,Y 330.006,Z 383.847,A -85,B 0,C 180,E1 16388.896,E2 16388.896} C_VEL
LIN {X 0,Y 330.011,Z 383.828,A -85,B 0,C 180,E1 16384.61,E2 16384.61} C_VEL
LIN {X 0,Y 330.017,Z 383.829,A -85,B 0,C 180,E1 16380.355,E2 16380.355} C_VEL
LIN {X 0,Y 329.998,Z 383.845,A -85,B 0,C 180,E1 16376.012,E2 16376.012} C_VEL
LIN {X 0,Y 329.99,Z 383.821,A -85,B 0,C 180,E1 16371.821,E2 16371.821} C_VEL
LIN {X 0,Y 329.987,Z 383.867,A -85,B 0,C 180,E1 16367.586,E2 16367.586} C_VEL
LIN {X 0,Y 329.976,Z 383.818,A -85,B 0,C 180,E1 16363.279,E2 16363.279} C_VEL
LIN {X 0,Y 329.986,Z 383.874,A -85,B 0,C 180,E1 16358.875,E2 16358.875} C_VEL
LIN {X 0,Y 329.992,Z 383.835,A -85,B 0,C 180,E1 16354.527,E2 16354.527} C_VEL
LIN {X 0,Y 330.014,Z 383.878,A -85,B 0,C 180,E1 16350.217,E2 16350.217} C_VEL
LIN {X 0,Y 330.06,Z 384.217,A -85,B 0,C 180,E1 16347.689,E2 16347.689} C_VEL
LIN {X 0,Y 330.451,Z 385.748,A -85,B 0,C 180,E1 16347.115,E2 16347.115} C_VEL
LIN {X 0,Y 332.165,Z 388.418,A -85,B 0,C 180,E1 16346.172,E2 16346.172} C_VEL
LIN {X 0,Y 335.13,Z 390.417,A -85,B 0,C 180,E1 16344.646,E2 16344.646} C_VEL
LIN {X 0,Y 336.182,Z 391.379,A -85,B 0,C 180,E1 16344.04,E2 16344.04} C_VEL
LIN {X 0,Y 338.255,Z 394.766,A -85,B 0,C 180,E1 16342.714,E2 16342.714} C_VEL
LIN {X 0,Y 341.305,Z 397.052,A -85,B 0,C 180,E1 16340.923,E2 16340.923} C_VEL
LIN {X 0,Y 342.593,Z 397.975,A -85,B 0,C 180,E1 16340.175,E2 16340.175} C_VEL
LIN {X 0,Y 344.611,Z 401.344,A -85,B 0,C 180,E1 16338.819,E2 16338.819} C_VEL
LIN {X 0,Y 347.832,Z 403.846,A -85,B 0,C 180,E1 16336.846,E2 16336.846} C_VEL
LIN {X 0,Y 349.027,Z 404.595,A -85,B 0,C 180,E1 16336.125,E2 16336.125} C_VEL
LIN {X 0,Y 351.474,Z 408.271,A -85,B 0,C 180,E1 16334.45,E2 16334.45} C_VEL
LIN {X 0,Y 354.331,Z 410.562,A -85,B 0,C 180,E1 16332.581,E2 16332.581} C_VEL
LIN {X 0,Y 355.849,Z 411.528,A -85,B 0,C 180,E1 16331.58,E2 16331.58} C_VEL
LIN {X 0,Y 358.029,Z 414.926,A -85,B 0,C 180,E1 16329.963,E2 16329.963} C_VEL
LIN {X 0,Y 361.295,Z 417.516,A -85,B 0,C 180,E1 16327.692,E2 16327.692} C_VEL
LIN {X 0,Y 362.751,Z 418.489,A -85,B 0,C 180,E1 16326.621,E2 16326.621} C_VEL
LIN {X 0,Y 364.918,Z 421.735,A -85,B 0,C 180,E1 16324.871,E2 16324.871} C_VEL
LIN {X 0,Y 367.84,Z 424.231,A -85,B 0,C 180,E1 16322.599,E2 16322.599} C_VEL
LIN {X 0,Y 370.003,Z 425.542,A -85,B 0,C 180,E1 16320.86,E2 16320.86} C_VEL
LIN {X 0,Y 372.238,Z 428.996,A -85,B 0,C 180,E1 16318.737,E2 16318.737} C_VEL
LIN {X 0,Y 375.105,Z 431.313,A -85,B 0,C 180,E1 16316.09,E2 16316.09} C_VEL
LIN {X 0,Y 377.391,Z 432.609,A -85,B 0,C 180,E1 16313.83,E2 16313.83} C_VEL
LIN {X 0,Y 379.183,Z 435.631,A -85,B 0,C 180,E1 16311.663,E2 16311.663} C_VEL
LIN {X 0,Y 381.613,Z 437.941,A -85,B 0,C 180,E1 16308.641,E2 16308.641} C_VEL
LIN {X 0,Y 384.046,Z 439.155,A -85,B 0,C 180,E1 16305.245,E2 16305.245} C_VEL
LIN {X 0,Y 385.43,Z 440.461,A -85,B 0,C 180,E1 16302.891,E2 16302.891} C_VEL
LIN {X 0,Y 386.684,Z 442.674,A -85,B 0,C 180,E1 16299.944,E2 16299.944} C_VEL
LIN {X 0,Y 387.711,Z 443.967,A -85,B 0,C 180,E1 16296.813,E2 16296.813} C_VEL
LIN {X 0,Y 388.465,Z 444.601,A -85,B 0,C 180,E1 16293.394,E2 16293.394} C_VEL
LIN {X 0,Y 388.714,Z 444.824,A -85,B 0,C 180,E1 16290,E2 16290} C_VEL
LIN {X 0,Y 388.465,Z 444.601,A -85,B 0,C 180,E1 16286.606,E2 16286.606} C_VEL
LIN {X 0,Y 387.711,Z 443.966,A -85,B 0,C 180,E1 16283.187,E2 16283.187} C_VEL
LIN {X 0,Y 386.668,Z 442.662,A -85,B 0,C 180,E1 16280.023,E2 16280.023} C_VEL
LIN {X 0,Y 385.429,Z 440.462,A -85,B 0,C 180,E1 16277.109,E2 16277.109} C_VEL
LIN {X 0,Y 384.046,Z 439.155,A -85,B 0,C 180,E1 16274.755,E2 16274.755} C_VEL
LIN {X 0,Y 381.614,Z 437.941,A -85,B 0,C 180,E1 16271.359,E2 16271.359} C_VEL
LIN {X 0,Y 379.183,Z 435.632,A -85,B 0,C 180,E1 16268.337,E2 16268.337} C_VEL
LIN {X 0,Y 377.008,Z 432.205,A -85,B 0,C 180,E1 16265.728,E2 16265.728} C_VEL
LIN {X 0,Y 373.704,Z 430.379,A -85,B 0,C 180,E1 16262.601,E2 16262.601} C_VEL
LIN {X 0,Y 371.055,Z 427.462,A -85,B 0,C 180,E1 16260.169,E2 16260.169} C_VEL
LIN {X 0,Y 369.731,Z 425.16,A -85,B 0,C 180,E1 16258.902,E2 16258.902} C_VEL
LIN {X 0,Y 366.225,Z 423.099,A -85,B 0,C 180,E1 16256.156,E2 16256.156} C_VEL
LIN {X 0,Y 363.28,Z 419.472,A -85,B 0,C 180,E1 16253.798,E2 16253.798} C_VEL
LIN {X 0,Y 362.414,Z 418.078,A -85,B 0,C 180,E1 16253.12,E2 16253.12} C_VEL
LIN {X 0,Y 358.793,Z 415.702,A -85,B 0,C 180,E1 16250.554,E2 16250.554} C_VEL
LIN {X 0,Y 356.295,Z 412.364,A -85,B 0,C 180,E1 16248.742,E2 16248.742} C_VEL
LIN {X 0,Y 355.487,Z 411.118,A -85,B 0,C 180,E1 16248.174,E2 16248.174} C_VEL
LIN {X 0,Y 352.15,Z 409.021,A -85,B 0,C 180,E1 16246.02,E2 16246.02} C_VEL
LIN {X 0,Y 349.392,Z 405.342,A -85,B 0,C 180,E1 16244.147,E2 16244.147} C_VEL
LIN {X 0,Y 348.763,Z 404.245,A -85,B 0,C 180,E1 16243.689,E2 16243.689} C_VEL
LIN {X 0,Y 345.202,Z 401.922,A -85,B 0,C 180,E1 16241.538,E2 16241.538} C_VEL
LIN {X 0,Y 343.002,Z 398.821,A -85,B 0,C 180,E1 16240.094,E2 16240.094} C_VEL
LIN {X 0,Y 342.156,Z 397.432,A -85,B 0,C 180,E1 16239.559,E2 16239.559} C_VEL
LIN {X 0,Y 338.841,Z 395.366,A -85,B 0,C 180,E1 16237.636,E2 16237.636} C_VEL
LIN {X 0,Y 336.67,Z 392.328,A -85,B 0,C 180,E1 16236.269,E2 16236.269} C_VEL
LIN {X 0,Y 335.754,Z 390.724,A -85,B 0,C 180,E1 16235.697,E2 16235.697} C_VEL
LIN {X 0,Y 332.331,Z 388.582,A -85,B 0,C 180,E1 16233.913,E2 16233.913} C_VEL
LIN {X 0,Y 330.522,Z 385.931,A -85,B 0,C 180,E1 16232.928,E2 16232.928} C_VEL
LIN {X 0,Y 330.078,Z 384.353,A -85,B 0,C 180,E1 16232.411,E2 16232.411} C_VEL
LIN {X 0,Y 329.986,Z 383.881,A -85,B 0,C 180,E1 16231.303,E2 16231.303} C_VEL
LIN {X 0,Y 329.983,Z 383.879,A -85,B 0,C 180,E1 16227.022,E2 16227.022} C_VEL
LIN {X 0,Y 330,Z 383.822,A -85,B 0,C 180,E1 16223.601,E2 16223.601} C_VEL
LIN {X 0,Y 328.983,Z 383.975,A -85,B 0,C 180,E1 16222.264,E2 16222.264} C_VEL
LIN {X 0,Y 324.107,Z 384.596,A -85,B 0,C 180,E1 16219.543,E2 16219.543} C_VEL
LIN {X 0,Y 322.125,Z 384.798,A -85,B 0,C 180,E1 16217.788,E2 16217.788} C_VEL
LIN {X 0,Y 322.058,Z 384.803,A -85,B 0,C 180,E1 16217.489,E2 16217.489} C_VEL
LIN {X 0,Y 322.057,Z 384.87,A -85,B 0,C 180,E1 16213.273,E2 16213.273} C_VEL
LIN {X 0,Y 322.04,Z 384.801,A -85,B 0,C 180,E1 16208.922,E2 16208.922} C_VEL
LIN {X 0,Y 322.045,Z 384.847,A -85,B 0,C 180,E1 16204.444,E2 16204.444} C_VEL
LIN {X 0,Y 322.044,Z 384.808,A -85,B 0,C 180,E1 16200.17,E2 16200.17} C_VEL
LIN {X 0,Y 322.057,Z 384.829,A -85,B 0,C 180,E1 16195.898,E2 16195.898} C_VEL
LIN {X 0,Y 322.07,Z 384.819,A -85,B 0,C 180,E1 16191.603,E2 16191.603} C_VEL
LIN {X 0,Y 322.075,Z 384.81,A -85,B 0,C 180,E1 16187.26,E2 16187.26} C_VEL
LIN {X 0,Y 322.068,Z 384.85,A -85,B 0,C 180,E1 16182.971,E2 16182.971} C_VEL
LIN {X 0,Y 322.052,Z 384.807,A -85,B 0,C 180,E1 16178.649,E2 16178.649} C_VEL
LIN {X 0,Y 322.049,Z 384.842,A -85,B 0,C 180,E1 16174.23,E2 16174.23} C_VEL
LIN {X 0,Y 322.098,Z 385.049,A -85,B 0,C 180,E1 16171.435,E2 16171.435} C_VEL
LIN {X 0,Y 322.33,Z 386.017,A -85,B 0,C 180,E1 16171.053,E2 16171.053} C_VEL
LIN {X 0,Y 324.004,Z 389.157,A -85,B 0,C 180,E1 16170.355,E2 16170.355} C_VEL
LIN {X 0,Y 327.078,Z 391.746,A -85,B 0,C 180,E1 16169.321,E2 16169.321} C_VEL
LIN {X 0,Y 329.479,Z 395.469,A -85,B 0,C 180,E1 16168.479,E2 16168.479} C_VEL
LIN {X 0,Y 332.578,Z 398.988,A -85,B 0,C 180,E1 16167.488,E2 16167.488} C_VEL
LIN {X 0,Y 338.361,Z 407.389,A -85,B 0,C 180,E1 16165.684,E2 16165.684} C_VEL
LIN {X 0,Y 343.197,Z 414.502,A -85,B 0,C 180,E1 16164.278,E2 16164.278} C_VEL
LIN {X 0,Y 350.687,Z 426.19,A -85,B 0,C 180,E1 16162.24,E2 16162.24} C_VEL
LIN {X 0,Y 359.515,Z 440.998,A -85,B 0,C 180,E1 16160.02,E2 16160.02} C_VEL
LIN {X 0,Y 368.866,Z 458.465,A -85,B 0,C 180,E1 16157.833,E2 16157.833} C_VEL
LIN {X 0,Y 372.826,Z 466.764,A -85,B 0,C 180,E1 16156.941,E2 16156.941} C_VEL
LIN {X 0,Y 364.57,Z 645.745,A -85,B 0,C 180,E1 16153.339,E2 16153.339} C_VEL
LIN {X 0,Y 362.608,Z 666.862,A -85,B 0,C 180,E1 16152.711,E2 16152.711} C_VEL
LIN {X 0,Y 360.109,Z 685.073,A -85,B 0,C 180,E1 16151.932,E2 16151.932} C_VEL
LIN {X 0,Y 357.551,Z 700.607,A -85,B 0,C 180,E1 16151.082,E2 16151.082} C_VEL
LIN {X 0,Y 354.33,Z 717.527,A -85,B 0,C 180,E1 16149.937,E2 16149.937} C_VEL
LIN {X 0,Y 350.068,Z 736.822,A -85,B 0,C 180,E1 16148.3,E2 16148.3} C_VEL
LIN {X 0,Y 346.296,Z 752.157,A -85,B 0,C 180,E1 16146.702,E2 16146.702} C_VEL
LIN {X 0,Y 342.315,Z 767.296,A -85,B 0,C 180,E1 16144.832,E2 16144.832} C_VEL
LIN {X 0,Y 337.744,Z 783.576,A -85,B 0,C 180,E1 16142.399,E2 16142.399} C_VEL
LIN {X 0,Y 334.054,Z 796.361,A -85,B 0,C 180,E1 16140.109,E2 16140.109} C_VEL
LIN {X 0,Y 330.572,Z 808.473,A -85,B 0,C 180,E1 16137.565,E2 16137.565} C_VEL
LIN {X 0,Y 326.992,Z 821.226,A -85,B 0,C 180,E1 16134.318,E2 16134.318} C_VEL
LIN {X 0,Y 324.597,Z 830.401,A -85,B 0,C 180,E1 16131.503,E2 16131.503} C_VEL
LIN {X 0,Y 322.564,Z 839.291,A -85,B 0,C 180,E1 16128.244,E2 16128.244} C_VEL
LIN {X 0,Y 321.136,Z 846.705,A -85,B 0,C 180,E1 16124.791,E2 16124.791} C_VEL
LIN {X 0,Y 320.401,Z 851.94,A -85,B 0,C 180,E1 16121.703,E2 16121.703} C_VEL
LIN {X 0,Y 320.056,Z 855.929,A -85,B 0,C 180,E1 16118.624,E2 16118.624} C_VEL
LIN {X 0,Y 319.948,Z 859.084,A -85,B 0,C 180,E1 16115.02,E2 16115.02} C_VEL
LIN {X 0,Y 319.96,Z 860.411,A -85,B 0,C 180,E1 16111.791,E2 16111.791} C_VEL
LIN {X 0,Y 319.967,Z 860.531,A -85,B 0,C 180,E1 16108.926,E2 16108.926} C_VEL
LIN {X 0,Y 319.949,Z 859.62,A -85,B 0,C 180,E1 16106.058,E2 16106.058} C_VEL
LIN {X 0,Y 319.975,Z 857.672,A -85,B 0,C 180,E1 16103.181,E2 16103.181} C_VEL
LIN {X 0,Y 320.201,Z 854.038,A -85,B 0,C 180,E1 16099.748,E2 16099.748} C_VEL
LIN {X 0,Y 320.872,Z 848.384,A -85,B 0,C 180,E1 16096.118,E2 16096.118} C_VEL
LIN {X 0,Y 321.937,Z 842.257,A -85,B 0,C 180,E1 16093.066,E2 16093.066} C_VEL
LIN {X 0,Y 323.724,Z 834.109,A -85,B 0,C 180,E1 16089.762,E2 16089.762} C_VEL
LIN {X 0,Y 326.358,Z 823.592,A -85,B 0,C 180,E1 16086.364,E2 16086.364} C_VEL
LIN {X 0,Y 329.1,Z 813.594,A -85,B 0,C 180,E1 16083.669,E2 16083.669} C_VEL
LIN {X 0,Y 332.657,Z 801.323,A -85,B 0,C 180,E1 16080.863,E2 16080.863} C_VEL
LIN {X 0,Y 336.739,Z 787.083,A -85,B 0,C 180,E1 16078.195,E2 16078.195} C_VEL
LIN {X 0,Y 340.34,Z 774.369,A -85,B 0,C 180,E1 16076.172,E2 16076.172} C_VEL
LIN {X 0,Y 344.666,Z 758.611,A -85,B 0,C 180,E1 16074.041,E2 16074.041} C_VEL
LIN {X 0,Y 348.913,Z 741.667,A -85,B 0,C 180,E1 16072.177,E2 16072.177} C_VEL
LIN {X 0,Y 352.269,Z 727.15,A -85,B 0,C 180,E1 16070.838,E2 16070.838} C_VEL
LIN {X 0,Y 355.6,Z 711.144,A -85,B 0,C 180,E1 16069.602,E2 16069.602} C_VEL
LIN {X 0,Y 359.336,Z 690.079,A -85,B 0,C 180,E1 16068.318,E2 16068.318} C_VEL
LIN {X 0,Y 361.857,Z 672.469,A -85,B 0,C 180,E1 16067.509,E2 16067.509} C_VEL
LIN {X 0,Y 363.905,Z 654.243,A -85,B 0,C 180,E1 16066.884,E2 16066.884} C_VEL
LIN {X 0,Y 365.561,Z 627.12,A -85,B 0,C 180,E1 16066.258,E2 16066.258} C_VEL
LIN {X 0,Y 372.746,Z 466.28,A -85,B 0,C 180,E1 16063.032,E2 16063.032} C_VEL
LIN {X 0,Y 363.343,Z 447.94,A -85,B 0,C 180,E1 16060.894,E2 16060.894} C_VEL
LIN {X 0,Y 354.383,Z 432.186,A -85,B 0,C 180,E1 16058.71,E2 16058.71} C_VEL
LIN {X 0,Y 347.391,Z 420.962,A -85,B 0,C 180,E1 16056.883,E2 16056.883} C_VEL
LIN {X 0,Y 339.985,Z 409.648,A -85,B 0,C 180,E1 16054.793,E2 16054.793} C_VEL
LIN {X 0,Y 335.669,Z 403.543,A -85,B 0,C 180,E1 16053.497,E2 16053.497} C_VEL
LIN {X 0,Y 330.684,Z 396.583,A -85,B 0,C 180,E1 16051.902,E2 16051.902} C_VEL
LIN {X 0,Y 327.88,Z 393.311,A -85,B 0,C 180,E1 16050.977,E2 16050.977} C_VEL
LIN {X 0,Y 326.687,Z 391.203,A -85,B 0,C 180,E1 16050.541,E2 16050.541} C_VEL
LIN {X 0,Y 323.675,Z 388.754,A -85,B 0,C 180,E1 16049.525,E2 16049.525} C_VEL
LIN {X 0,Y 322.172,Z 385.392,A -85,B 0,C 180,E1 16048.76,E2 16048.76} C_VEL
LIN {X 0,Y 322.044,Z 384.815,A -85,B 0,C 180,E1 16047.964,E2 16047.964} C_VEL
LIN {X 0,Y 322.048,Z 384.839,A -85,B 0,C 180,E1 16043.616,E2 16043.616} C_VEL
LIN {X 0,Y 322.06,Z 384.833,A -85,B 0,C 180,E1 16039.22,E2 16039.22} C_VEL
LIN {X 0,Y 322.085,Z 384.799,A -85,B 0,C 180,E1 16034.754,E2 16034.754} C_VEL
LIN {X 0,Y 322.065,Z 384.868,A -85,B 0,C 180,E1 16030.229,E2 16030.229} C_VEL
LIN {X 0,Y 322.044,Z 384.8,A -85,B 0,C 180,E1 16025.888,E2 16025.888} C_VEL
LIN {X 0,Y 322.045,Z 384.851,A -85,B 0,C 180,E1 16021.431,E2 16021.431} C_VEL
LIN {X 0,Y 322.047,Z 384.809,A -85,B 0,C 180,E1 16016.982,E2 16016.982} C_VEL
LIN {X 0,Y 322.061,Z 384.825,A -85,B 0,C 180,E1 16012.695,E2 16012.695} C_VEL
LIN {X 0,Y 322.072,Z 384.825,A -85,B 0,C 180,E1 16008.367,E2 16008.367} C_VEL
LIN {X 0,Y 322.076,Z 384.808,A -85,B 0,C 180,E1 16004.155,E2 16004.155} C_VEL
LIN {X 0,Y 322.07,Z 384.859,A -85,B 0,C 180,E1 15999.853,E2 15999.853} C_VEL
LIN {X 0,Y 322.054,Z 384.81,A -85,B 0,C 180,E1 15995.622,E2 15995.622} C_VEL
LIN {X 0,Y 322.055,Z 384.905,A -85,B 0,C 180,E1 15991.246,E2 15991.246} C_VEL
LIN {X 0,Y 322.161,Z 385.523,A -85,B 0,C 180,E1 15990.646,E2 15990.646} C_VEL
LIN {X 0,Y 324.062,Z 389.24,A -85,B 0,C 180,E1 15989.562,E2 15989.562} C_VEL
LIN {X 0,Y 326.963,Z 391.298,A -85,B 0,C 180,E1 15988.277,E2 15988.277} C_VEL
LIN {X 0,Y 327.939,Z 392.186,A -85,B 0,C 180,E1 15987.817,E2 15987.817} C_VEL
LIN {X 0,Y 329.805,Z 395.284,A -85,B 0,C 180,E1 15986.835,E2 15986.835} C_VEL
LIN {X 0,Y 332.617,Z 397.676,A -85,B 0,C 180,E1 15985.391,E2 15985.391} C_VEL
LIN {X 0,Y 334.339,Z 398.729,A -85,B 0,C 180,E1 15984.497,E2 15984.497} C_VEL
LIN {X 0,Y 336.728,Z 402.427,A -85,B 0,C 180,E1 15983.009,E2 15983.009} C_VEL
LIN {X 0,Y 339.805,Z 404.79,A -85,B 0,C 180,E1 15981.203,E2 15981.203} C_VEL
LIN {X 0,Y 340.917,Z 405.589,A -85,B 0,C 180,E1 15980.541,E2 15980.541} C_VEL
LIN {X 0,Y 343.189,Z 409.098,A -85,B 0,C 180,E1 15979.054,E2 15979.054} C_VEL
LIN {X 0,Y 346.416,Z 411.62,A -85,B 0,C 180,E1 15977.079,E2 15977.079} C_VEL
LIN {X 0,Y 347.62,Z 412.513,A -85,B 0,C 180,E1 15976.359,E2 15976.359} C_VEL
LIN {X 0,Y 350.366,Z 416.331,A -85,B 0,C 180,E1 15974.499,E2 15974.499} C_VEL
LIN {X 0,Y 353.532,Z 418.638,A -85,B 0,C 180,E1 15972.44,E2 15972.44} C_VEL
LIN {X 0,Y 354.447,Z 419.386,A -85,B 0,C 180,E1 15971.82,E2 15971.82} C_VEL
LIN {X 0,Y 356.796,Z 422.82,A -85,B 0,C 180,E1 15970.106,E2 15970.106} C_VEL
LIN {X 0,Y 360.031,Z 425.352,A -85,B 0,C 180,E1 15967.86,E2 15967.86} C_VEL
LIN {X 0,Y 361.414,Z 426.335,A -85,B 0,C 180,E1 15966.851,E2 15966.851} C_VEL
LIN {X 0,Y 363.718,Z 429.614,A -85,B 0,C 180,E1 15965.013,E2 15965.013} C_VEL
LIN {X 0,Y 366.498,Z 432.011,A -85,B 0,C 180,E1 15962.851,E2 15962.851} C_VEL
LIN {X 0,Y 368.752,Z 433.402,A -85,B 0,C 180,E1 15961.058,E2 15961.058} C_VEL
LIN {X 0,Y 371.077,Z 436.847,A -85,B 0,C 180,E1 15958.893,E2 15958.893} C_VEL
LIN {X 0,Y 373.802,Z 439.114,A -85,B 0,C 180,E1 15956.36,E2 15956.36} C_VEL
LIN {X 0,Y 376.286,Z 440.555,A -85,B 0,C 180,E1 15953.952,E2 15953.952} C_VEL
LIN {X 0,Y 378.136,Z 443.581,A -85,B 0,C 180,E1 15951.726,E2 15951.726} C_VEL
LIN {X 0,Y 380.592,Z 445.87,A -85,B 0,C 180,E1 15948.693,E2 15948.693} C_VEL
LIN {X 0,Y 383.039,Z 447.086,A -85,B 0,C 180,E1 15945.286,E2 15945.286} C_VEL
LIN {X 0,Y 384.337,Z 448.286,A -85,B 0,C 180,E1 15943.081,E2 15943.081} C_VEL
LIN {X 0,Y 385.606,Z 450.536,A -85,B 0,C 180,E1 15940.155,E2 15940.155} C_VEL
LIN {X 0,Y 386.696,Z 451.877,A -85,B 0,C 180,E1 15936.926,E2 15936.926} C_VEL
LIN {X 0,Y 387.457,Z 452.522,A -85,B 0,C 180,E1 15933.551,E2 15933.551} C_VEL
LIN {X 0,Y 387.727,Z 452.755,A -85,B 0,C 180,E1 15930.148,E2 15930.148} C_VEL
LIN {X 0,Y 387.503,Z 452.552,A -85,B 0,C 180,E1 15926.733,E2 15926.733} C_VEL
LIN {X 0,Y 386.78,Z 451.951,A -85,B 0,C 180,E1 15923.32,E2 15923.32} C_VEL
LIN {X 0,Y 385.751,Z 450.668,A -85,B 0,C 180,E1 15920.15,E2 15920.15} C_VEL
LIN {X 0,Y 384.505,Z 448.591,A -85,B 0,C 180,E1 15917.231,E2 15917.231} C_VEL
LIN {X 0,Y 383.252,Z 447.191,A -85,B 0,C 180,E1 15915.032,E2 15915.032} C_VEL
LIN {X 0,Y 380.965,Z 446.106,A -85,B 0,C 180,E1 15911.787,E2 15911.787} C_VEL
LIN {X 0,Y 378.573,Z 444.068,A -85,B 0,C 180,E1 15908.77,E2 15908.77} C_VEL
LIN {X 0,Y 376.605,Z 441.195,A -85,B 0,C 180,E1 15906.45,E2 15906.45} C_VEL
LIN {X 0,Y 375.733,Z 440.054,A -85,B 0,C 180,E1 15905.473,E2 15905.473} C_VEL
LIN {X 0,Y 372.418,Z 438.12,A -85,B 0,C 180,E1 15902.325,E2 15902.325} C_VEL
LIN {X 0,Y 369.745,Z 435.162,A -85,B 0,C 180,E1 15899.901,E2 15899.901} C_VEL
LIN {X 0,Y 368.314,Z 432.944,A -85,B 0,C 180,E1 15898.587,E2 15898.587} C_VEL
LIN {X 0,Y 364.81,Z 430.732,A -85,B 0,C 180,E1 15895.817,E2 15895.817} C_VEL
LIN {X 0,Y 361.854,Z 427.131,A -85,B 0,C 180,E1 15893.504,E2 15893.504} C_VEL
LIN {X 0,Y 361.056,Z 425.873,A -85,B 0,C 180,E1 15892.866,E2 15892.866} C_VEL
LIN {X 0,Y 357.512,Z 423.535,A -85,B 0,C 180,E1 15890.385,E2 15890.385} C_VEL
LIN {X 0,Y 354.778,Z 419.996,A -85,B 0,C 180,E1 15888.424,E2 15888.424} C_VEL
LIN {X 0,Y 354.109,Z 418.91,A -85,B 0,C 180,E1 15887.939,E2 15887.939} C_VEL
LIN {X 0,Y 350.635,Z 416.619,A -85,B 0,C 180,E1 15885.684,E2 15885.684} C_VEL
LIN {X 0,Y 347.754,Z 412.761,A -85,B 0,C 180,E1 15883.734,E2 15883.734} C_VEL
LIN {X 0,Y 347.03,Z 411.912,A -85,B 0,C 180,E1 15883.279,E2 15883.279} C_VEL
LIN {X 0,Y 343.479,Z 409.394,A -85,B 0,C 180,E1 15881.125,E2 15881.125} C_VEL
LIN {X 0,Y 341.12,Z 406,A -85,B 0,C 180,E1 15879.594,E2 15879.594} C_VEL
LIN {X 0,Y 340.407,Z 405.081,A -85,B 0,C 180,E1 15879.149,E2 15879.149} C_VEL
LIN {X 0,Y 337.101,Z 402.826,A -85,B 0,C 180,E1 15877.222,E2 15877.222} C_VEL
LIN {X 0,Y 334.75,Z 399.524,A -85,B 0,C 180,E1 15875.768,E2 15875.768} C_VEL
LIN {X 0,Y 333.953,Z 398.322,A -85,B 0,C 180,E1 15875.287,E2 15875.287} C_VEL
LIN {X 0,Y 330.613,Z 396.171,A -85,B 0,C 180,E1 15873.591,E2 15873.591} C_VEL
LIN {X 0,Y 328.317,Z 393.051,A -85,B 0,C 180,E1 15872.399,E2 15872.399} C_VEL
LIN {X 0,Y 327.346,Z 391.458,A -85,B 0,C 180,E1 15871.885,E2 15871.885} C_VEL
LIN {X 0,Y 324.342,Z 389.544,A -85,B 0,C 180,E1 15870.563,E2 15870.563} C_VEL
LIN {X 0,Y 322.396,Z 386.358,A -85,B 0,C 180,E1 15869.611,E2 15869.611} C_VEL
LIN {X 0,Y 322.063,Z 384.988,A -85,B 0,C 180,E1 15869.007,E2 15869.007} C_VEL
LIN {X 0,Y 322.047,Z 384.812,A -85,B 0,C 180,E1 15864.543,E2 15864.543} C_VEL
LIN {X 0,Y 322.059,Z 384.866,A -85,B 0,C 180,E1 15860.338,E2 15860.338} C_VEL
LIN {X 0,Y 322.058,Z 384.803,A -85,B 0,C 180,E1 15857.489,E2 15857.489} C_VEL
LIN {X 0,Y 321.036,Z 384.941,A -85,B 0,C 180,E1 15856.119,E2 15856.119} C_VEL
LIN {X 0,Y 316.313,Z 385.585,A -85,B 0,C 180,E1 15853.428,E2 15853.428} C_VEL
LIN {X 0,Y 314.217,Z 385.803,A -85,B 0,C 180,E1 15851.632,E2 15851.632} C_VEL
LIN {X 0,Y 314.112,Z 385.804,A -85,B 0,C 180,E1 15851.223,E2 15851.223} C_VEL
LIN {X 0,Y 314.102,Z 385.83,A -85,B 0,C 180,E1 15846.716,E2 15846.716} C_VEL
LIN {X 0,Y 314.1,Z 385.788,A -85,B 0,C 180,E1 15842.364,E2 15842.364} C_VEL
LIN {X 0,Y 314.12,Z 385.854,A -85,B 0,C 180,E1 15837.986,E2 15837.986} C_VEL
LIN {X 0,Y 314.141,Z 385.781,A -85,B 0,C 180,E1 15833.413,E2 15833.413} C_VEL
LIN {X 0,Y 314.125,Z 385.844,A -85,B 0,C 180,E1 15828.983,E2 15828.983} C_VEL
LIN {X 0,Y 314.105,Z 385.8,A -85,B 0,C 180,E1 15824.484,E2 15824.484} C_VEL
LIN {X 0,Y 314.105,Z 385.807,A -85,B 0,C 180,E1 15820.079,E2 15820.079} C_VEL
LIN {X 0,Y 314.116,Z 385.845,A -85,B 0,C 180,E1 15815.75,E2 15815.75} C_VEL
LIN {X 0,Y 314.144,Z 386.067,A -85,B 0,C 180,E1 15814.141,E2 15814.141} C_VEL
LIN {X 0,Y 314.524,Z 387.52,A -85,B 0,C 180,E1 15813.611,E2 15813.611} C_VEL
LIN {X 0,Y 316.534,Z 390.595,A -85,B 0,C 180,E1 15812.734,E2 15812.734} C_VEL
LIN {X 0,Y 319.355,Z 392.717,A -85,B 0,C 180,E1 15811.678,E2 15811.678} C_VEL
LIN {X 0,Y 321.62,Z 396.421,A -85,B 0,C 180,E1 15810.779,E2 15810.779} C_VEL
LIN {X 0,Y 324.397,Z 399.018,A -85,B 0,C 180,E1 15809.809,E2 15809.809} C_VEL
LIN {X 0,Y 327.371,Z 403.086,A -85,B 0,C 180,E1 15808.765,E2 15808.765} C_VEL
LIN {X 0,Y 330.636,Z 407.325,A -85,B 0,C 180,E1 15807.684,E2 15807.684} C_VEL
LIN {X 0,Y 338.804,Z 419.234,A -85,B 0,C 180,E1 15805.145,E2 15805.145} C_VEL
LIN {X 0,Y 347.222,Z 432.73,A -85,B 0,C 180,E1 15802.76,E2 15802.76} C_VEL
LIN {X 0,Y 355.509,Z 446.91,A -85,B 0,C 180,E1 15800.607,E2 15800.607} C_VEL
LIN {X 0,Y 364.436,Z 463.87,A -85,B 0,C 180,E1 15798.446,E2 15798.446} C_VEL
LIN {X 0,Y 367.22,Z 469.983,A -85,B 0,C 180,E1 15797.787,E2 15797.787} C_VEL
LIN {X 0,Y 358.778,Z 645.459,A -85,B 0,C 180,E1 15794.219,E2 15794.219} C_VEL
LIN {X 0,Y 356.747,Z 666.624,A -85,B 0,C 180,E1 15793.586,E2 15793.586} C_VEL
LIN {X 0,Y 354.075,Z 685.379,A -85,B 0,C 180,E1 15792.775,E2 15792.775} C_VEL
LIN {X 0,Y 351.282,Z 701.613,A -85,B 0,C 180,E1 15791.87,E2 15791.87} C_VEL
LIN {X 0,Y 347.524,Z 720.444,A -85,B 0,C 180,E1 15790.557,E2 15790.557} C_VEL
LIN {X 0,Y 343.325,Z 738.197,A -85,B 0,C 180,E1 15788.979,E2 15788.979} C_VEL
LIN {X 0,Y 339.426,Z 753.341,A -85,B 0,C 180,E1 15787.359,E2 15787.359} C_VEL
LIN {X 0,Y 334.769,Z 770.193,A -85,B 0,C 180,E1 15785.199,E2 15785.199} C_VEL
LIN {X 0,Y 330.434,Z 784.713,A -85,B 0,C 180,E1 15782.923,E2 15782.923} C_VEL
LIN {X 0,Y 326.78,Z 796.782,A -85,B 0,C 180,E1 15780.7,E2 15780.7} C_VEL
LIN {X 0,Y 322.859,Z 809.811,A -85,B 0,C 180,E1 15777.88,E2 15777.88} C_VEL
LIN {X 0,Y 319.362,Z 821.512,A -85,B 0,C 180,E1 15774.769,E2 15774.769} C_VEL
LIN {X 0,Y 316.863,Z 830.567,A -85,B 0,C 180,E1 15771.908,E2 15771.908} C_VEL
LIN {X 0,Y 314.593,Z 839.919,A -85,B 0,C 180,E1 15768.339,E2 15768.339} C_VEL
LIN {X 0,Y 313.191,Z 846.8,A -85,B 0,C 180,E1 15764.986,E2 15764.986} C_VEL
LIN {X 0,Y 312.418,Z 851.972,A -85,B 0,C 180,E1 15761.819,E2 15761.819} C_VEL
LIN {X 0,Y 312.032,Z 856.319,A -85,B 0,C 180,E1 15758.29,E2 15758.29} C_VEL
LIN {X 0,Y 311.947,Z 859.115,A -85,B 0,C 180,E1 15754.596,E2 15754.596} C_VEL
LIN {X 0,Y 311.965,Z 860.205,A -85,B 0,C 180,E1 15751.653,E2 15751.653} C_VEL
LIN {X 0,Y 311.969,Z 860.265,A -85,B 0,C 180,E1 15748.715,E2 15748.715} C_VEL
LIN {X 0,Y 311.948,Z 859.294,A -85,B 0,C 180,E1 15745.772,E2 15745.772} C_VEL
LIN {X 0,Y 312.001,Z 857.136,A -85,B 0,C 180,E1 15742.635,E2 15742.635} C_VEL
LIN {X 0,Y 312.33,Z 852.788,A -85,B 0,C 180,E1 15738.739,E2 15738.739} C_VEL
LIN {X 0,Y 313.073,Z 847.472,A -85,B 0,C 180,E1 15735.387,E2 15735.387} C_VEL
LIN {X 0,Y 314.311,Z 841.126,A -85,B 0,C 180,E1 15732.219,E2 15732.219} C_VEL
LIN {X 0,Y 316.554,Z 831.79,A -85,B 0,C 180,E1 15728.507,E2 15728.507} C_VEL
LIN {X 0,Y 319.039,Z 822.647,A -85,B 0,C 180,E1 15725.564,E2 15725.564} C_VEL
LIN {X 0,Y 321.97,Z 812.647,A -85,B 0,C 180,E1 15722.839,E2 15722.839} C_VEL
LIN {X 0,Y 326.025,Z 799.338,A -85,B 0,C 180,E1 15719.805,E2 15719.805} C_VEL
LIN {X 0,Y 329.949,Z 786.34,A -85,B 0,C 180,E1 15717.358,E2 15717.358} C_VEL
LIN {X 0,Y 333.742,Z 773.565,A -85,B 0,C 180,E1 15715.305,E2 15715.305} C_VEL
LIN {X 0,Y 338.501,Z 756.904,A -85,B 0,C 180,E1 15713.053,E2 15713.053} C_VEL
LIN {X 0,Y 342.726,Z 740.62,A -85,B 0,C 180,E1 15711.262,E2 15711.262} C_VEL
LIN {X 0,Y 346.233,Z 725.989,A -85,B 0,C 180,E1 15709.912,E2 15709.912} C_VEL
LIN {X 0,Y 350,Z 708.452,A -85,B 0,C 180,E1 15708.566,E2 15708.566} C_VEL
LIN {X 0,Y 353.597,Z 688.353,A -85,B 0,C 180,E1 15707.374,E2 15707.374} C_VEL
LIN {X 0,Y 356.099,Z 671.316,A -85,B 0,C 180,E1 15706.599,E2 15706.599} C_VEL
LIN {X 0,Y 358.394,Z 651.106,A -85,B 0,C 180,E1 15705.918,E2 15705.918} C_VEL
LIN {X 0,Y 360.22,Z 617.834,A -85,B 0,C 180,E1 15705.191,E2 15705.191} C_VEL
LIN {X 0,Y 367.121,Z 469.316,A -85,B 0,C 180,E1 15702.177,E2 15702.177} C_VEL
LIN {X 0,Y 358.108,Z 451.664,A -85,B 0,C 180,E1 15700.038,E2 15700.038} C_VEL
LIN {X 0,Y 348.676,Z 435.034,A -85,B 0,C 180,E1 15697.627,E2 15697.627} C_VEL
LIN {X 0,Y 340.986,Z 422.727,A -85,B 0,C 180,E1 15695.498,E2 15695.498} C_VEL
LIN {X 0,Y 336.137,Z 415.383,A -85,B 0,C 180,E1 15694.059,E2 15694.059} C_VEL
LIN {X 0,Y 328.899,Z 404.802,A -85,B 0,C 180,E1 15691.737,E2 15691.737} C_VEL
LIN {X 0,Y 324.769,Z 399.699,A -85,B 0,C 180,E1 15690.331,E2 15690.331} C_VEL
LIN {X 0,Y 323.668,Z 398.174,A -85,B 0,C 180,E1 15689.934,E2 15689.934} C_VEL
LIN {X 0,Y 320.654,Z 395.182,A -85,B 0,C 180,E1 15688.858,E2 15688.858} C_VEL
LIN {X 0,Y 318.933,Z 392.213,A -85,B 0,C 180,E1 15688.159,E2 15688.159} C_VEL
LIN {X 0,Y 315.919,Z 389.921,A -85,B 0,C 180,E1 15687.018,E2 15687.018} C_VEL
LIN {X 0,Y 314.251,Z 386.613,A -85,B 0,C 180,E1 15686.153,E2 15686.153} C_VEL
LIN {X 0,Y 314.121,Z 385.86,A -85,B 0,C 180,E1 15685.456,E2 15685.456} C_VEL
LIN {X 0,Y 314.129,Z 385.793,A -85,B 0,C 180,E1 15681.087,E2 15681.087} C_VEL
LIN {X 0,Y 314.137,Z 385.823,A -85,B 0,C 180,E1 15676.653,E2 15676.653} C_VEL
LIN {X 0,Y 314.121,Z 385.808,A -85,B 0,C 180,E1 15672.268,E2 15672.268} C_VEL
LIN {X 0,Y 314.111,Z 385.8,A -85,B 0,C 180,E1 15668.059,E2 15668.059} C_VEL
LIN {X 0,Y 314.104,Z 385.831,A -85,B 0,C 180,E1 15663.658,E2 15663.658} C_VEL
LIN {X 0,Y 314.1,Z 385.788,A -85,B 0,C 180,E1 15659.278,E2 15659.278} C_VEL
LIN {X 0,Y 314.118,Z 385.853,A -85,B 0,C 180,E1 15654.895,E2 15654.895} C_VEL
LIN {X 0,Y 314.126,Z 385.783,A -85,B 0,C 180,E1 15650.482,E2 15650.482} C_VEL
